   // GB2[6869] := 16#D1C5;
   // GB2[6870] := 16#BCAF;
   // GB2[6871] := 16#B9CD;
   // GB2[6872] := 16#EFF4;
   // GB2[6873] := 16#B4C6;
   // GB2[6874] := 16#D3BA;
   // GB2[6875] := 16#F6C2;
   // GB2[6876] := 16#B3FB;
   // GB2[6877] := 16#F6C3;
   // GB2[6878] := 16#B5F1;
   // GB2[6879] := 16#F6C5;
   // GB2[6880] := 16#D3EA;
   // GB2[6881] := 16#F6A7;
   // GB2[6882] := 16#D1A9;
   // GB2[6883] := 16#F6A9;
   // GB2[6884] := 16#F6A8;
   // GB2[6885] := 16#C1E3;
   // GB2[6886] := 16#C0D7;
   // GB2[6887] := 16#B1A2;
   // GB2[6888] := 16#CEED;
   // GB2[6889] := 16#D0E8;
   // GB2[6890] := 16#F6AB;
   // GB2[6891] := 16#CFF6;
   // GB2[6892] := 16#F6AA;
   // GB2[6893] := 16#D5F0;
   // GB2[6894] := 16#F6AC;
   // GB2[6895] := 16#C3B9;
   // GB2[6896] := 16#BBF4;
   // GB2[6897] := 16#F6AE;
   // GB2[6898] := 16#F6AD;
   // GB2[6899] := 16#C4DE;
   // GB2[6900] := 16#C1D8;
   // GB2[6901] := 16#CBAA;
   // GB2[6902] := 16#CFBC;
   // GB2[6903] := 16#F6AF;
   // GB2[6904] := 16#F6B0;
   // GB2[6905] := 16#F6B1;
   // GB2[6906] := 16#C2B6;
   // GB2[6907] := 16#B0D4;
   // GB2[6908] := 16#C5F9;
   // GB2[6909] := 16#F6B2;
   // GB2[6910] := 16#C7E0;
   // GB2[6911] := 16#F6A6;
   // GB2[6912] := 16#BEB8;
   // GB2[6913] := 16#BEB2;
   // GB2[6914] := 16#B5E5;
   // GB2[6915] := 16#B7C7;
   // GB2[6916] := 16#BFBF;
   // GB2[6917] := 16#C3D2;
   // GB2[6918] := 16#C3E6;
   // GB2[6919] := 16#D8CC;
   // GB2[6920] := 16#B8EF;
   // GB2[6921] := 16#BDF9;
   // GB2[6922] := 16#D1A5;
   // GB2[6923] := 16#B0D0;
   // GB2[6924] := 16#F7B0;
   // GB2[6925] := 16#F7B1;
   // GB2[6926] := 16#D0AC;
   // GB2[6927] := 16#B0B0;
   // GB2[6928] := 16#F7B2;
   // GB2[6929] := 16#F7B3;
   // GB2[6930] := 16#F7B4;
   // GB2[6931] := 16#C7CA;
   // GB2[6932] := 16#BECF;
   // GB2[6933] := 16#F7B7;
   // GB2[6934] := 16#F7B6;
   // GB2[6935] := 16#B1DE;
   // GB2[6936] := 16#F7B5;
   // GB2[6937] := 16#F7B8;
   // GB2[6938] := 16#F7B9;
   // GB2[6939] := 16#CEA4;
   // GB2[6940] := 16#C8CD;
   // GB2[6941] := 16#BAAB;
   // GB2[6942] := 16#E8B8;
   // GB2[6943] := 16#E8B9;
   // GB2[6944] := 16#E8BA;
   // GB2[6945] := 16#BEC2;
   // GB2[6946] := 16#D2F4;
   // GB2[6947] := 16#D4CF;
   // GB2[6948] := 16#C9D8;
   // GB2[6949] := 16#D2B3;
   // GB2[6950] := 16#B6A5;
   // GB2[6951] := 16#C7EA;
   // GB2[6952] := 16#F1FC;
   // GB2[6953] := 16#CFEE;
   // GB2[6954] := 16#CBB3;
   // GB2[6955] := 16#D0EB;
   // GB2[6956] := 16#E7EF;
   // GB2[6957] := 16#CDE7;
   // GB2[6958] := 16#B9CB;
   // GB2[6959] := 16#B6D9;
   // GB2[6960] := 16#F1FD;
   // GB2[6961] := 16#B0E4;
   // GB2[6962] := 16#CBCC;
   // GB2[6963] := 16#F1FE;
   // GB2[6964] := 16#D4A4;
   // GB2[6965] := 16#C2AD;
   // GB2[6966] := 16#C1EC;
   // GB2[6967] := 16#C6C4;
   // GB2[6968] := 16#BEB1;
   // GB2[6969] := 16#F2A1;
   // GB2[6970] := 16#BCD5;
   // GB2[6971] := 16#F2A2;
   // GB2[6972] := 16#F2A3;
   // GB2[6973] := 16#F2A4;
   // GB2[6974] := 16#D2C3;
   // GB2[6975] := 16#C6B5;
   // GB2[6976] := 16#CDC7;
   // GB2[6977] := 16#F2A5;
   // GB2[6978] := 16#D3B1;
   // GB2[6979] := 16#BFC5;
   // GB2[6980] := 16#CCE2;
   // GB2[6981] := 16#F2A6;
   // GB2[6982] := 16#F2A7;
   // GB2[6983] := 16#D1D5;
   // GB2[6984] := 16#B6EE;
   // GB2[6985] := 16#F2A8;
   // GB2[6986] := 16#F2A9;
   // GB2[6987] := 16#B5DF;
   // GB2[6988] := 16#F2AA;
   // GB2[6989] := 16#F2AB;
   // GB2[6990] := 16#B2FC;
   // GB2[6991] := 16#F2AC;
   // GB2[6992] := 16#F2AD;
   // GB2[6993] := 16#C8A7;
   // GB2[6994] := 16#B7E7;
   // GB2[6995] := 16#ECA9;
   // GB2[6996] := 16#ECAA;
   // GB2[6997] := 16#ECAB;
   // GB2[6998] := 16#ECAC;
   // GB2[6999] := 16#C6AE;
   // GB2[7000] := 16#ECAD;
   // GB2[7001] := 16#ECAE;
   // GB2[7002] := 16#B7C9;
   // GB2[7003] := 16#CAB3;
   // GB2[7004] := 16#E2B8;
   // GB2[7005] := 16#F7CF;
   // GB2[7006] := 16#F7D0;
   // GB2[7007] := 16#B2CD;
   // GB2[7008] := 16#F7D1;
   // GB2[7009] := 16#F7D3;
   // GB2[7010] := 16#F7D2;
   // GB2[7011] := 16#E2BB;
   // GB2[7012] := 16#BCA2;
   // GB2[7013] := 16#E2BC;
   // GB2[7014] := 16#E2BD;
   // GB2[7015] := 16#E2BE;
   // GB2[7016] := 16#E2BF;
   // GB2[7017] := 16#E2C0;
   // GB2[7018] := 16#E2C1;
   // GB2[7019] := 16#B7B9;
   // GB2[7020] := 16#D2FB;
   // GB2[7021] := 16#BDA4;
   // GB2[7022] := 16#CACE;
   // GB2[7023] := 16#B1A5;
   // GB2[7024] := 16#CBC7;
   // GB2[7025] := 16#E2C2;
   // GB2[7026] := 16#B6FC;
   // GB2[7027] := 16#C8C4;
   // GB2[7028] := 16#E2C3;
   // GB2[7029] := 16#BDC8;
   // GB2[7030] := 16#B1FD;
   // GB2[7031] := 16#E2C4;
   // GB2[7032] := 16#B6F6;
   // GB2[7033] := 16#E2C5;
   // GB2[7034] := 16#C4D9;
   // GB2[7035] := 16#E2C6;
   // GB2[7036] := 16#CFDA;
   // GB2[7037] := 16#B9DD;
   // GB2[7038] := 16#E2C7;
   // GB2[7039] := 16#C0A1;
   // GB2[7040] := 16#E2C8;
   // GB2[7041] := 16#B2F6;
   // GB2[7042] := 16#E2C9;
   // GB2[7043] := 16#C1F3;
   // GB2[7044] := 16#E2CA;
   // GB2[7045] := 16#E2CB;
   // GB2[7046] := 16#C2F8;
   // GB2[7047] := 16#E2CC;
   // GB2[7048] := 16#E2CD;
   // GB2[7049] := 16#E2CE;
   // GB2[7050] := 16#CAD7;
   // GB2[7051] := 16#D8B8;
   // GB2[7052] := 16#D9E5;
   // GB2[7053] := 16#CFE3;
   // GB2[7054] := 16#F0A5;
   // GB2[7055] := 16#DCB0;
   // GB2[7056] := 16#C2ED;
   // GB2[7057] := 16#D4A6;
   // GB2[7058] := 16#CDD4;
   // GB2[7059] := 16#D1B1;
   // GB2[7060] := 16#B3DB;
   // GB2[7061] := 16#C7FD;
   // GB2[7062] := 16#B2B5;
   // GB2[7063] := 16#C2BF;
   // GB2[7064] := 16#E6E0;
   // GB2[7065] := 16#CABB;
   // GB2[7066] := 16#E6E1;
   // GB2[7067] := 16#E6E2;
   // GB2[7068] := 16#BED4;
   // GB2[7069] := 16#E6E3;
   // GB2[7070] := 16#D7A4;
   // GB2[7071] := 16#CDD5;
   // GB2[7072] := 16#E6E5;
   // GB2[7073] := 16#BCDD;
   // GB2[7074] := 16#E6E4;
   // GB2[7075] := 16#E6E6;
   // GB2[7076] := 16#E6E7;
   // GB2[7077] := 16#C2EE;
   // GB2[7078] := 16#BDBE;
   // GB2[7079] := 16#E6E8;
   // GB2[7080] := 16#C2E6;
   // GB2[7081] := 16#BAA7;
   // GB2[7082] := 16#E6E9;
   // GB2[7083] := 16#E6EA;
   // GB2[7084] := 16#B3D2;
   // GB2[7085] := 16#D1E9;
   // GB2[7086] := 16#BFA5;
   // GB2[7087] := 16#E6EB;
   // GB2[7088] := 16#C6EF;
   // GB2[7089] := 16#E6EC;
   // GB2[7090] := 16#E6ED;
   // GB2[7091] := 16#E6EE;
   // GB2[7092] := 16#C6AD;
   // GB2[7093] := 16#E6EF;
   // GB2[7094] := 16#C9A7;
   // GB2[7095] := 16#E6F0;
   // GB2[7096] := 16#E6F1;
   // GB2[7097] := 16#E6F2;
   // GB2[7098] := 16#E5B9;
   // GB2[7099] := 16#E6F3;
   // GB2[7100] := 16#E6F4;
   // GB2[7101] := 16#C2E2;
   // GB2[7102] := 16#E6F5;
   // GB2[7103] := 16#E6F6;
   // GB2[7104] := 16#D6E8;
   // GB2[7105] := 16#E6F7;
   // GB2[7106] := 16#E6F8;
   // GB2[7107] := 16#B9C7;
   // GB2[7108] := 16#F7BB;
   // GB2[7109] := 16#F7BA;
   // GB2[7110] := 16#F7BE;
   // GB2[7111] := 16#F7BC;
   // GB2[7112] := 16#BAA1;
   // GB2[7113] := 16#F7BF;
   // GB2[7114] := 16#F7C0;
   // GB2[7115] := 16#F7C2;
   // GB2[7116] := 16#F7C1;
   // GB2[7117] := 16#F7C4;
   // GB2[7118] := 16#F7C3;
   // GB2[7119] := 16#F7C5;
   // GB2[7120] := 16#F7C6;
   // GB2[7121] := 16#F7C7;
   // GB2[7122] := 16#CBE8;
   // GB2[7123] := 16#B8DF;
   // GB2[7124] := 16#F7D4;
   // GB2[7125] := 16#F7D5;
   // GB2[7126] := 16#F7D6;
   // GB2[7127] := 16#F7D8;
   // GB2[7128] := 16#F7DA;
   // GB2[7129] := 16#F7D7;
   // GB2[7130] := 16#F7DB;
   // GB2[7131] := 16#F7D9;
   // GB2[7132] := 16#D7D7;
   // GB2[7133] := 16#F7DC;
   // GB2[7134] := 16#F7DD;
   // GB2[7135] := 16#F7DE;
   // GB2[7136] := 16#F7DF;
   // GB2[7137] := 16#F7E0;
   // GB2[7138] := 16#DBCB;
   // GB2[7139] := 16#D8AA;
   // GB2[7140] := 16#E5F7;
   // GB2[7141] := 16#B9ED;
   // GB2[7142] := 16#BFFD;
   // GB2[7143] := 16#BBEA;
   // GB2[7144] := 16#F7C9;
   // GB2[7145] := 16#C6C7;
   // GB2[7146] := 16#F7C8;
   // GB2[7147] := 16#F7CA;
   // GB2[7148] := 16#F7CC;
   // GB2[7149] := 16#F7CB;
   // GB2[7150] := 16#F7CD;
   // GB2[7151] := 16#CEBA;
   // GB2[7152] := 16#F7CE;
   // GB2[7153] := 16#C4A7;
   // GB2[7154] := 16#D3E3;
   // GB2[7155] := 16#F6CF;
   // GB2[7156] := 16#C2B3;
   // GB2[7157] := 16#F6D0;
   // GB2[7158] := 16#F6D1;
   // GB2[7159] := 16#F6D2;
   // GB2[7160] := 16#F6D3;
   // GB2[7161] := 16#F6D4;
   // GB2[7162] := 16#F6D6;
   // GB2[7163] := 16#B1AB;
   // GB2[7164] := 16#F6D7;
   // GB2[7165] := 16#F6D8;
   // GB2[7166] := 16#F6D9;
   // GB2[7167] := 16#F6DA;
   // GB2[7168] := 16#F6DB;
   // GB2[7169] := 16#F6DC;
   // GB2[7170] := 16#F6DD;
   // GB2[7171] := 16#F6DE;
   // GB2[7172] := 16#CFCA;
   // GB2[7173] := 16#F6DF;
   // GB2[7174] := 16#F6E0;
   // GB2[7175] := 16#F6E1;
   // GB2[7176] := 16#F6E2;
   // GB2[7177] := 16#F6E3;
   // GB2[7178] := 16#F6E4;
   // GB2[7179] := 16#C0F0;
   // GB2[7180] := 16#F6E5;
   // GB2[7181] := 16#F6E6;
   // GB2[7182] := 16#F6E7;
   // GB2[7183] := 16#F6E8;
   // GB2[7184] := 16#F6E9;
   // GB2[7185] := 16#F6EA;
   // GB2[7186] := 16#F6EB;
   // GB2[7187] := 16#F6EC;
   // GB2[7188] := 16#F6ED;
   // GB2[7189] := 16#F6EE;
   // GB2[7190] := 16#F6EF;
   // GB2[7191] := 16#F6F0;
   // GB2[7192] := 16#F6F1;
   // GB2[7193] := 16#F6F2;
   // GB2[7194] := 16#F6F3;
   // GB2[7195] := 16#F6F4;
   // GB2[7196] := 16#BEA8;
   // GB2[7197] := 16#F6F5;
   // GB2[7198] := 16#F6F6;
   // GB2[7199] := 16#F6F7;
   // GB2[7200] := 16#F6F8;
   // GB2[7201] := 16#C8FA;
   // GB2[7202] := 16#F6F9;
   // GB2[7203] := 16#F6FA;
   // GB2[7204] := 16#F6FB;
   // GB2[7205] := 16#F6FC;
   // GB2[7206] := 16#F6FD;
   // GB2[7207] := 16#F6FE;
   // GB2[7208] := 16#F7A1;
   // GB2[7209] := 16#F7A2;
   // GB2[7210] := 16#F7A3;
   // GB2[7211] := 16#F7A4;
   // GB2[7212] := 16#F7A5;
   // GB2[7213] := 16#F7A6;
   // GB2[7214] := 16#F7A7;
   // GB2[7215] := 16#F7A8;
   // GB2[7216] := 16#B1EE;
   // GB2[7217] := 16#F7A9;
   // GB2[7218] := 16#F7AA;
   // GB2[7219] := 16#F7AB;
   // GB2[7220] := 16#F7AC;
   // GB2[7221] := 16#F7AD;
   // GB2[7222] := 16#C1DB;
   // GB2[7223] := 16#F7AE;
   // GB2[7224] := 16#F7AF;
   // GB2[7225] := 16#C4F1;
   // GB2[7226] := 16#F0AF;
   // GB2[7227] := 16#BCA6;
   // GB2[7228] := 16#F0B0;
   // GB2[7229] := 16#C3F9;
   // GB2[7230] := 16#C5B8;
   // GB2[7231] := 16#D1BB;
   // GB2[7232] := 16#F0B1;
   // GB2[7233] := 16#F0B2;
   // GB2[7234] := 16#F0B3;
   // GB2[7235] := 16#F0B4;
   // GB2[7236] := 16#F0B5;
   // GB2[7237] := 16#D1BC;
   // GB2[7238] := 16#D1EC;
   // GB2[7239] := 16#F0B7;
   // GB2[7240] := 16#F0B6;
   // GB2[7241] := 16#D4A7;
   // GB2[7242] := 16#CDD2;
   // GB2[7243] := 16#F0B8;
   // GB2[7244] := 16#F0BA;
   // GB2[7245] := 16#F0B9;
   // GB2[7246] := 16#F0BB;
   // GB2[7247] := 16#F0BC;
   // GB2[7248] := 16#B8EB;
   // GB2[7249] := 16#F0BD;
   // GB2[7250] := 16#BAE8;
   // GB2[7251] := 16#F0BE;
   // GB2[7252] := 16#F0BF;
   // GB2[7253] := 16#BEE9;
   // GB2[7254] := 16#F0C0;
   // GB2[7255] := 16#B6EC;
   // GB2[7256] := 16#F0C1;
   // GB2[7257] := 16#F0C2;
   // GB2[7258] := 16#F0C3;
   // GB2[7259] := 16#F0C4;
   // GB2[7260] := 16#C8B5;
   // GB2[7261] := 16#F0C5;
   // GB2[7262] := 16#F0C6;
   // GB2[7263] := 16#F0C7;
   // GB2[7264] := 16#C5F4;
   // GB2[7265] := 16#F0C8;
   // GB2[7266] := 16#F0C9;
   // GB2[7267] := 16#F0CA;
   // GB2[7268] := 16#F7BD;
   // GB2[7269] := 16#F0CB;
   // GB2[7270] := 16#F0CC;
   // GB2[7271] := 16#F0CD;
   // GB2[7272] := 16#F0CE;
   // GB2[7273] := 16#F0CF;
   // GB2[7274] := 16#BAD7;
   // GB2[7275] := 16#F0D0;
   // GB2[7276] := 16#F0D1;
   // GB2[7277] := 16#F0D2;
   // GB2[7278] := 16#F0D3;
   // GB2[7279] := 16#F0D4;
   // GB2[7280] := 16#F0D5;
   // GB2[7281] := 16#F0D6;
   // GB2[7282] := 16#F0D8;
   // GB2[7283] := 16#D3A5;
   // GB2[7284] := 16#F0D7;
   // GB2[7285] := 16#F0D9;
   // GB2[7286] := 16#F5BA;
   // GB2[7287] := 16#C2B9;
   // GB2[7288] := 16#F7E4;
   // GB2[7289] := 16#F7E5;
   // GB2[7290] := 16#F7E6;
   // GB2[7291] := 16#F7E7;
   // GB2[7292] := 16#F7E8;
   // GB2[7293] := 16#C2B4;
   // GB2[7294] := 16#F7EA;
   // GB2[7295] := 16#F7EB;
   // GB2[7296] := 16#C2F3;
   // GB2[7297] := 16#F4F0;
   // GB2[7298] := 16#F4EF;
   // GB2[7299] := 16#C2E9;
   // GB2[7300] := 16#F7E1;
   // GB2[7301] := 16#F7E2;
   // GB2[7302] := 16#BBC6;
   // GB2[7303] := 16#D9E4;
   // GB2[7304] := 16#CAF2;
   // GB2[7305] := 16#C0E8;
   // GB2[7306] := 16#F0A4;
   // GB2[7307] := 16#BADA;
   // GB2[7308] := 16#C7AD;
   // GB2[7309] := 16#C4AC;
   // GB2[7310] := 16#F7EC;
   // GB2[7311] := 16#F7ED;
   // GB2[7312] := 16#F7EE;
   // GB2[7313] := 16#F7F0;
   // GB2[7314] := 16#F7EF;
   // GB2[7315] := 16#F7F1;
   // GB2[7316] := 16#F7F4;
   // GB2[7317] := 16#F7F3;
   // GB2[7318] := 16#F7F2;
   // GB2[7319] := 16#F7F5;
   // GB2[7320] := 16#F7F6;
   // GB2[7321] := 16#EDE9;
   // GB2[7322] := 16#EDEA;
   // GB2[7323] := 16#EDEB;
   // GB2[7324] := 16#F6BC;
   // GB2[7325] := 16#F6BD;
   // GB2[7326] := 16#F6BE;
   // GB2[7327] := 16#B6A6;
   // GB2[7328] := 16#D8BE;
   // GB2[7329] := 16#B9C4;
   // GB2[7330] := 16#D8BB;
   // GB2[7331] := 16#DCB1;
   // GB2[7332] := 16#CAF3;
   // GB2[7333] := 16#F7F7;
   // GB2[7334] := 16#F7F8;
   // GB2[7335] := 16#F7F9;
   // GB2[7336] := 16#F7FB;
   // GB2[7337] := 16#F7FA;
   // GB2[7338] := 16#B1C7;
   // GB2[7339] := 16#F7FC;
   // GB2[7340] := 16#F7FD;
   // GB2[7341] := 16#F7FE;
   // GB2[7342] := 16#C6EB;
   // GB2[7343] := 16#ECB4;
   // GB2[7344] := 16#B3DD;
   // GB2[7345] := 16#F6B3;
   // GB2[7346] := 16#F6B4;
   // GB2[7347] := 16#C1E4;
   // GB2[7348] := 16#F6B5;
   // GB2[7349] := 16#F6B6;
   // GB2[7350] := 16#F6B7;
   // GB2[7351] := 16#F6B8;
   // GB2[7352] := 16#F6B9;
   // GB2[7353] := 16#F6BA;
   // GB2[7354] := 16#C8A3;
   // GB2[7355] := 16#F6BB;
   // GB2[7356] := 16#C1FA;
   // GB2[7357] := 16#B9A8;
   // GB2[7358] := 16#EDE8;
   // GB2[7359] := 16#B9EA;
   // GB2[7360] := 16#D9DF;
   // GB2[7361] := 16#A6F2;
   // GB2[7362] := 16#A6F4;
   // GB2[7363] := 16#A6F5;
   // GB2[7364] := 16#A6E0;
   // GB2[7365] := 16#A6E1;
   // GB2[7366] := 16#A6F0;
   // GB2[7367] := 16#A6F1;
   // GB2[7368] := 16#A6E2;
   // GB2[7369] := 16#A6E3;
   // GB2[7370] := 16#A6EE;
   // GB2[7371] := 16#A6EF;
   // GB2[7372] := 16#A6E6;
   // GB2[7373] := 16#A6E7;
   // GB2[7374] := 16#A6E4;
   // GB2[7375] := 16#A6E5;
   // GB2[7376] := 16#A6E8;
   // GB2[7377] := 16#A6E9;
   // GB2[7378] := 16#A6EA;
   // GB2[7379] := 16#A6EB;
   // GB2[7380] := 16#A3A1;
   // GB2[7381] := 16#A3A2;
   // GB2[7382] := 16#A3A3;
   // GB2[7383] := 16#A1E7;
   // GB2[7384] := 16#A3A5;
   // GB2[7385] := 16#A3A6;
   // GB2[7386] := 16#A3A7;
   // GB2[7387] := 16#A3A8;
   // GB2[7388] := 16#A3A9;
   // GB2[7389] := 16#A3AA;
   // GB2[7390] := 16#A3AB;
   // GB2[7391] := 16#A3AC;
   // GB2[7392] := 16#A3AD;
   // GB2[7393] := 16#A3AE;
   // GB2[7394] := 16#A3AF;
   // GB2[7395] := 16#A3B0;
   // GB2[7396] := 16#A3B1;
   // GB2[7397] := 16#A3B2;
   // GB2[7398] := 16#A3B3;
   // GB2[7399] := 16#A3B4;
   // GB2[7400] := 16#A3B5;
   // GB2[7401] := 16#A3B6;
   // GB2[7402] := 16#A3B7;
   // GB2[7403] := 16#A3B8;
   // GB2[7404] := 16#A3B9;
   // GB2[7405] := 16#A3BA;
   // GB2[7406] := 16#A3BB;
   // GB2[7407] := 16#A3BC;
   // GB2[7408] := 16#A3BD;
   // GB2[7409] := 16#A3BE;
   // GB2[7410] := 16#A3BF;
   // GB2[7411] := 16#A3C0;
   // GB2[7412] := 16#A3C1;
   // GB2[7413] := 16#A3C2;
   // GB2[7414] := 16#A3C3;
   // GB2[7415] := 16#A3C4;
   // GB2[7416] := 16#A3C5;
   // GB2[7417] := 16#A3C6;
   // GB2[7418] := 16#A3C7;
   // GB2[7419] := 16#A3C8;
   // GB2[7420] := 16#A3C9;
   // GB2[7421] := 16#A3CA;
   // GB2[7422] := 16#A3CB;
   // GB2[7423] := 16#A3CC;
   // GB2[7424] := 16#A3CD;
   // GB2[7425] := 16#A3CE;
   // GB2[7426] := 16#A3CF;
   // GB2[7427] := 16#A3D0;
   // GB2[7428] := 16#A3D1;
   // GB2[7429] := 16#A3D2;
   // GB2[7430] := 16#A3D3;
   // GB2[7431] := 16#A3D4;
   // GB2[7432] := 16#A3D5;
   // GB2[7433] := 16#A3D6;
   // GB2[7434] := 16#A3D7;
   // GB2[7435] := 16#A3D8;
   // GB2[7436] := 16#A3D9;
   // GB2[7437] := 16#A3DA;
   // GB2[7438] := 16#A3DB;
   // GB2[7439] := 16#A3DC;
   // GB2[7440] := 16#A3DD;
   // GB2[7441] := 16#A3DE;
   // GB2[7442] := 16#A3DF;
   // GB2[7443] := 16#A3E0;
   // GB2[7444] := 16#A3E1;
   // GB2[7445] := 16#A3E2;
   // GB2[7446] := 16#A3E3;
   // GB2[7447] := 16#A3E4;
   // GB2[7448] := 16#A3E5;
   // GB2[7449] := 16#A3E6;
   // GB2[7450] := 16#A3E7;
   // GB2[7451] := 16#A3E8;
   // GB2[7452] := 16#A3E9;
   // GB2[7453] := 16#A3EA;
   // GB2[7454] := 16#A3EB;
   // GB2[7455] := 16#A3EC;
   // GB2[7456] := 16#A3ED;
   // GB2[7457] := 16#A3EE;
   // GB2[7458] := 16#A3EF;
   // GB2[7459] := 16#A3F0;
   // GB2[7460] := 16#A3F1;
   // GB2[7461] := 16#A3F2;
   // GB2[7462] := 16#A3F3;
   // GB2[7463] := 16#A3F4;
   // GB2[7464] := 16#A3F5;
   // GB2[7465] := 16#A3F6;
   // GB2[7466] := 16#A3F7;
   // GB2[7467] := 16#A3F8;
   // GB2[7468] := 16#A3F9;
   // GB2[7469] := 16#A3FA;
   // GB2[7470] := 16#A3FB;
   // GB2[7471] := 16#A3FC;
   // GB2[7472] := 16#A3FD;
   // GB2[7473] := 16#A1AB;
   // GB2[7474] := 16#A1E9;
   // GB2[7475] := 16#A1EA;
   // GB2[7476] := 16#A3FE;
   // GB2[7477] := 16#A3A4;
   // GB2[7478] := 0;
   // GB2[7479] := 0;
BEGIN
   IF #UNICODE < 16#0080 THEN
       #GB2312 := #UNICODE;
   ELSE
       #hi := 7480;
       #li := 0;
       FOR #j := 0 TO 13 BY 1 DO
           #i := #li + (#hi - #li) / 2;
           IF #UNICODE = #UNI[#i] THEN
               #GB2312 := #GB2[#i];
               EXIT;
           END_IF;
           IF #UNICODE > #UNI[#i] THEN
               #li := #i;
           ELSE
               #hi := #i;
           END_IF;
       END_FOR;
   END_IF;
END_FUNCTION_BLOCK

// ===== library: MasterCopy "UNI_TO_GBK" =====

// folder: FB/UNICODE_FB

FUNCTION_BLOCK "UNI_TO_GBK"   // FB1, SCL
{ S7_Optimized_Access := 'TRUE' }
VERSION : 0.1
   VAR_INPUT
      UNICODE : Word;
   END_VAR
   VAR_OUTPUT
      GBK : Word;
   END_VAR
   VAR
      UNICODE_TO_GBK : Array[0..43592] of Word;
   END_VAR
   VAR_TEMP
      i : UDInt;
      j : UDInt;
      li : UDInt;
      hi : UDInt;
   END_VAR
   // UNICODE_TO_GBK[0] := 16#00A4;
   // UNICODE_TO_GBK[1] := 16#A1E8;
   // UNICODE_TO_GBK[2] := 16#00A7;
   // UNICODE_TO_GBK[3] := 16#A1EC;
   // UNICODE_TO_GBK[4] := 16#00A8;
   // UNICODE_TO_GBK[5] := 16#A1A7;
   // UNICODE_TO_GBK[6] := 16#00B0;
   // UNICODE_TO_GBK[7] := 16#A1E3;
   // UNICODE_TO_GBK[8] := 16#00B1;
   // UNICODE_TO_GBK[9] := 16#A1C0;
   // UNICODE_TO_GBK[10] := 16#00B7;
   // UNICODE_TO_GBK[11] := 16#A1A4;
   // UNICODE_TO_GBK[12] := 16#00D7;
   // UNICODE_TO_GBK[13] := 16#A1C1;
   // UNICODE_TO_GBK[14] := 16#00E0;
   // UNICODE_TO_GBK[15] := 16#A8A4;
   // UNICODE_TO_GBK[16] := 16#00E1;
   // UNICODE_TO_GBK[17] := 16#A8A2;
   // UNICODE_TO_GBK[18] := 16#00E8;
   // UNICODE_TO_GBK[19] := 16#A8A8;
   // UNICODE_TO_GBK[20] := 16#00E9;
   // UNICODE_TO_GBK[21] := 16#A8A6;
   // UNICODE_TO_GBK[22] := 16#00EA;
   // UNICODE_TO_GBK[23] := 16#A8BA;
   // UNICODE_TO_GBK[24] := 16#00EC;
   // UNICODE_TO_GBK[25] := 16#A8AC;
   // UNICODE_TO_GBK[26] := 16#00ED;
   // UNICODE_TO_GBK[27] := 16#A8AA;
   // UNICODE_TO_GBK[28] := 16#00F2;
   // UNICODE_TO_GBK[29] := 16#A8B0;
   // UNICODE_TO_GBK[30] := 16#00F3;
   // UNICODE_TO_GBK[31] := 16#A8AE;
   // UNICODE_TO_GBK[32] := 16#00F7;
   // UNICODE_TO_GBK[33] := 16#A1C2;
   // UNICODE_TO_GBK[34] := 16#00F9;
   // UNICODE_TO_GBK[35] := 16#A8B4;
   // UNICODE_TO_GBK[36] := 16#00FA;
   // UNICODE_TO_GBK[37] := 16#A8B2;
   // UNICODE_TO_GBK[38] := 16#00FC;
   // UNICODE_TO_GBK[39] := 16#A8B9;
   // UNICODE_TO_GBK[40] := 16#0101;
   // UNICODE_TO_GBK[41] := 16#A8A1;
   // UNICODE_TO_GBK[42] := 16#0113;
   // UNICODE_TO_GBK[43] := 16#A8A5;
   // UNICODE_TO_GBK[44] := 16#011B;
   // UNICODE_TO_GBK[45] := 16#A8A7;
   // UNICODE_TO_GBK[46] := 16#012B;
   // UNICODE_TO_GBK[47] := 16#A8A9;
   // UNICODE_TO_GBK[48] := 16#0144;
   // UNICODE_TO_GBK[49] := 16#A8BD;
   // UNICODE_TO_GBK[50] := 16#0148;
   // UNICODE_TO_GBK[51] := 16#A8BE;
   // UNICODE_TO_GBK[52] := 16#014D;
   // UNICODE_TO_GBK[53] := 16#A8AD;
   // UNICODE_TO_GBK[54] := 16#016B;
   // UNICODE_TO_GBK[55] := 16#A8B1;
   // UNICODE_TO_GBK[56] := 16#01CE;
   // UNICODE_TO_GBK[57] := 16#A8A3;
   // UNICODE_TO_GBK[58] := 16#01D0;
   // UNICODE_TO_GBK[59] := 16#A8AB;
   // UNICODE_TO_GBK[60] := 16#01D2;
   // UNICODE_TO_GBK[61] := 16#A8AF;
   // UNICODE_TO_GBK[62] := 16#01D4;
   // UNICODE_TO_GBK[63] := 16#A8B3;
   // UNICODE_TO_GBK[64] := 16#01D6;
   // UNICODE_TO_GBK[65] := 16#A8B5;
   // UNICODE_TO_GBK[66] := 16#01D8;
   // UNICODE_TO_GBK[67] := 16#A8B6;
   // UNICODE_TO_GBK[68] := 16#01DA;
   // UNICODE_TO_GBK[69] := 16#A8B7;
   // UNICODE_TO_GBK[70] := 16#01DC;
   // UNICODE_TO_GBK[71] := 16#A8B8;
   // UNICODE_TO_GBK[72] := 16#0251;
   // UNICODE_TO_GBK[73] := 16#A8BB;
   // UNICODE_TO_GBK[74] := 16#0261;
   // UNICODE_TO_GBK[75] := 16#A8C0;
   // UNICODE_TO_GBK[76] := 16#02C7;
   // UNICODE_TO_GBK[77] := 16#A1A6;
   // UNICODE_TO_GBK[78] := 16#02C9;
   // UNICODE_TO_GBK[79] := 16#A1A5;
   // UNICODE_TO_GBK[80] := 16#02CA;
   // UNICODE_TO_GBK[81] := 16#A840;
   // UNICODE_TO_GBK[82] := 16#02CB;
   // UNICODE_TO_GBK[83] := 16#A841;
   // UNICODE_TO_GBK[84] := 16#02D9;
   // UNICODE_TO_GBK[85] := 16#A842;
   // UNICODE_TO_GBK[86] := 16#0391;
   // UNICODE_TO_GBK[87] := 16#A6A1;
   // UNICODE_TO_GBK[88] := 16#0392;
   // UNICODE_TO_GBK[89] := 16#A6A2;
   // UNICODE_TO_GBK[90] := 16#0393;
   // UNICODE_TO_GBK[91] := 16#A6A3;
   // UNICODE_TO_GBK[92] := 16#0394;
   // UNICODE_TO_GBK[93] := 16#A6A4;
   // UNICODE_TO_GBK[94] := 16#0395;
   // UNICODE_TO_GBK[95] := 16#A6A5;
   // UNICODE_TO_GBK[96] := 16#0396;
   // UNICODE_TO_GBK[97] := 16#A6A6;
   // UNICODE_TO_GBK[98] := 16#0397;
   // UNICODE_TO_GBK[99] := 16#A6A7;
   // UNICODE_TO_GBK[100] := 16#0398;
   // UNICODE_TO_GBK[101] := 16#A6A8;
   // UNICODE_TO_GBK[102] := 16#0399;
   // UNICODE_TO_GBK[103] := 16#A6A9;
   // UNICODE_TO_GBK[104] := 16#039A;
   // UNICODE_TO_GBK[105] := 16#A6AA;
   // UNICODE_TO_GBK[106] := 16#039B;
   // UNICODE_TO_GBK[107] := 16#A6AB;
   // UNICODE_TO_GBK[108] := 16#039C;
   // UNICODE_TO_GBK[109] := 16#A6AC;
   // UNICODE_TO_GBK[110] := 16#039D;
   // UNICODE_TO_GBK[111] := 16#A6AD;
   // UNICODE_TO_GBK[112] := 16#039E;
   // UNICODE_TO_GBK[113] := 16#A6AE;
   // UNICODE_TO_GBK[114] := 16#039F;
   // UNICODE_TO_GBK[115] := 16#A6AF;
   // UNICODE_TO_GBK[116] := 16#03A0;
   // UNICODE_TO_GBK[117] := 16#A6B0;
   // UNICODE_TO_GBK[118] := 16#03A1;
   // UNICODE_TO_GBK[119] := 16#A6B1;
   // UNICODE_TO_GBK[120] := 16#03A3;
   // UNICODE_TO_GBK[121] := 16#A6B2;
   // UNICODE_TO_GBK[122] := 16#03A4;
   // UNICODE_TO_GBK[123] := 16#A6B3;
   // UNICODE_TO_GBK[124] := 16#03A5;
   // UNICODE_TO_GBK[125] := 16#A6B4;
   // UNICODE_TO_GBK[126] := 16#03A6;
   // UNICODE_TO_GBK[127] := 16#A6B5;
   // UNICODE_TO_GBK[128] := 16#03A7;
   // UNICODE_TO_GBK[129] := 16#A6B6;
   // UNICODE_TO_GBK[130] := 16#03A8;
   // UNICODE_TO_GBK[131] := 16#A6B7;
   // UNICODE_TO_GBK[132] := 16#03A9;
   // UNICODE_TO_GBK[133] := 16#A6B8;
   // UNICODE_TO_GBK[134] := 16#03B1;
   // UNICODE_TO_GBK[135] := 16#A6C1;
   // UNICODE_TO_GBK[136] := 16#03B2;
   // UNICODE_TO_GBK[137] := 16#A6C2;
   // UNICODE_TO_GBK[138] := 16#03B3;
   // UNICODE_TO_GBK[139] := 16#A6C3;
   // UNICODE_TO_GBK[140] := 16#03B4;
   // UNICODE_TO_GBK[141] := 16#A6C4;
   // UNICODE_TO_GBK[142] := 16#03B5;
   // UNICODE_TO_GBK[143] := 16#A6C5;
   // UNICODE_TO_GBK[144] := 16#03B6;
   // UNICODE_TO_GBK[145] := 16#A6C6;
   // UNICODE_TO_GBK[146] := 16#03B7;
   // UNICODE_TO_GBK[147] := 16#A6C7;
   // UNICODE_TO_GBK[148] := 16#03B8;
   // UNICODE_TO_GBK[149] := 16#A6C8;
   // UNICODE_TO_GBK[150] := 16#03B9;
   // UNICODE_TO_GBK[151] := 16#A6C9;
   // UNICODE_TO_GBK[152] := 16#03BA;
   // UNICODE_TO_GBK[153] := 16#A6CA;
   // UNICODE_TO_GBK[154] := 16#03BB;
   // UNICODE_TO_GBK[155] := 16#A6CB;
   // UNICODE_TO_GBK[156] := 16#03BC;
   // UNICODE_TO_GBK[157] := 16#A6CC;
   // UNICODE_TO_GBK[158] := 16#03BD;
   // UNICODE_TO_GBK[159] := 16#A6CD;
   // UNICODE_TO_GBK[160] := 16#03BE;
   // UNICODE_TO_GBK[161] := 16#A6CE;
   // UNICODE_TO_GBK[162] := 16#03BF;
   // UNICODE_TO_GBK[163] := 16#A6CF;
   // UNICODE_TO_GBK[164] := 16#03C0;
   // UNICODE_TO_GBK[165] := 16#A6D0;
   // UNICODE_TO_GBK[166] := 16#03C1;
   // UNICODE_TO_GBK[167] := 16#A6D1;
   // UNICODE_TO_GBK[168] := 16#03C3;
   // UNICODE_TO_GBK[169] := 16#A6D2;
   // UNICODE_TO_GBK[170] := 16#03C4;
   // UNICODE_TO_GBK[171] := 16#A6D3;
   // UNICODE_TO_GBK[172] := 16#03C5;
   // UNICODE_TO_GBK[173] := 16#A6D4;
   // UNICODE_TO_GBK[174] := 16#03C6;
   // UNICODE_TO_GBK[175] := 16#A6D5;
   // UNICODE_TO_GBK[176] := 16#03C7;
   // UNICODE_TO_GBK[177] := 16#A6D6;
   // UNICODE_TO_GBK[178] := 16#03C8;
   // UNICODE_TO_GBK[179] := 16#A6D7;
   // UNICODE_TO_GBK[180] := 16#03C9;
   // UNICODE_TO_GBK[181] := 16#A6D8;
   // UNICODE_TO_GBK[182] := 16#0401;
   // UNICODE_TO_GBK[183] := 16#A7A7;
   // UNICODE_TO_GBK[184] := 16#0410;
   // UNICODE_TO_GBK[185] := 16#A7A1;
   // UNICODE_TO_GBK[186] := 16#0411;
   // UNICODE_TO_GBK[187] := 16#A7A2;
   // UNICODE_TO_GBK[188] := 16#0412;
   // UNICODE_TO_GBK[189] := 16#A7A3;
   // UNICODE_TO_GBK[190] := 16#0413;
   // UNICODE_TO_GBK[191] := 16#A7A4;
   // UNICODE_TO_GBK[192] := 16#0414;
   // UNICODE_TO_GBK[193] := 16#A7A5;
   // UNICODE_TO_GBK[194] := 16#0415;
   // UNICODE_TO_GBK[195] := 16#A7A6;
   // UNICODE_TO_GBK[196] := 16#0416;
   // UNICODE_TO_GBK[197] := 16#A7A8;
   // UNICODE_TO_GBK[198] := 16#0417;
   // UNICODE_TO_GBK[199] := 16#A7A9;
   // UNICODE_TO_GBK[200] := 16#0418;
   // UNICODE_TO_GBK[201] := 16#A7AA;
   // UNICODE_TO_GBK[202] := 16#0419;
   // UNICODE_TO_GBK[203] := 16#A7AB;
   // UNICODE_TO_GBK[204] := 16#041A;
   // UNICODE_TO_GBK[205] := 16#A7AC;
   // UNICODE_TO_GBK[206] := 16#041B;
   // UNICODE_TO_GBK[207] := 16#A7AD;
   // UNICODE_TO_GBK[208] := 16#041C;
   // UNICODE_TO_GBK[209] := 16#A7AE;
   // UNICODE_TO_GBK[210] := 16#041D;
   // UNICODE_TO_GBK[211] := 16#A7AF;
   // UNICODE_TO_GBK[212] := 16#041E;
   // UNICODE_TO_GBK[213] := 16#A7B0;
   // UNICODE_TO_GBK[214] := 16#041F;
   // UNICODE_TO_GBK[215] := 16#A7B1;
   // UNICODE_TO_GBK[216] := 16#0420;
   // UNICODE_TO_GBK[217] := 16#A7B2;
   // UNICODE_TO_GBK[218] := 16#0421;
   // UNICODE_TO_GBK[219] := 16#A7B3;
   // UNICODE_TO_GBK[220] := 16#0422;
   // UNICODE_TO_GBK[221] := 16#A7B4;
   // UNICODE_TO_GBK[222] := 16#0423;
   // UNICODE_TO_GBK[223] := 16#A7B5;
   // UNICODE_TO_GBK[224] := 16#0424;
   // UNICODE_TO_GBK[225] := 16#A7B6;
   // UNICODE_TO_GBK[226] := 16#0425;
   // UNICODE_TO_GBK[227] := 16#A7B7;
   // UNICODE_TO_GBK[228] := 16#0426;
   // UNICODE_TO_GBK[229] := 16#A7B8;
   // UNICODE_TO_GBK[230] := 16#0427;
   // UNICODE_TO_GBK[231] := 16#A7B9;
   // UNICODE_TO_GBK[232] := 16#0428;
   // UNICODE_TO_GBK[233] := 16#A7BA;
   // UNICODE_TO_GBK[234] := 16#0429;
   // UNICODE_TO_GBK[235] := 16#A7BB;
   // UNICODE_TO_GBK[236] := 16#042A;
   // UNICODE_TO_GBK[237] := 16#A7BC;
   // UNICODE_TO_GBK[238] := 16#042B;
   // UNICODE_TO_GBK[239] := 16#A7BD;
   // UNICODE_TO_GBK[240] := 16#042C;
   // UNICODE_TO_GBK[241] := 16#A7BE;
   // UNICODE_TO_GBK[242] := 16#042D;
   // UNICODE_TO_GBK[243] := 16#A7BF;
   // UNICODE_TO_GBK[244] := 16#042E;
   // UNICODE_TO_GBK[245] := 16#A7C0;
   // UNICODE_TO_GBK[246] := 16#042F;
   // UNICODE_TO_GBK[247] := 16#A7C1;
   // UNICODE_TO_GBK[248] := 16#0430;
   // UNICODE_TO_GBK[249] := 16#A7D1;
   // UNICODE_TO_GBK[250] := 16#0431;
   // UNICODE_TO_GBK[251] := 16#A7D2;
   // UNICODE_TO_GBK[252] := 16#0432;
   // UNICODE_TO_GBK[253] := 16#A7D3;
   // UNICODE_TO_GBK[254] := 16#0433;
   // UNICODE_TO_GBK[255] := 16#A7D4;
   // UNICODE_TO_GBK[256] := 16#0434;
   // UNICODE_TO_GBK[257] := 16#A7D5;
   // UNICODE_TO_GBK[258] := 16#0435;
   // UNICODE_TO_GBK[259] := 16#A7D6;
   // UNICODE_TO_GBK[260] := 16#0436;
   // UNICODE_TO_GBK[261] := 16#A7D8;
   // UNICODE_TO_GBK[262] := 16#0437;
   // UNICODE_TO_GBK[263] := 16#A7D9;
   // UNICODE_TO_GBK[264] := 16#0438;
   // UNICODE_TO_GBK[265] := 16#A7DA;
   // UNICODE_TO_GBK[266] := 16#0439;
   // UNICODE_TO_GBK[267] := 16#A7DB;
   // UNICODE_TO_GBK[268] := 16#043A;
   // UNICODE_TO_GBK[269] := 16#A7DC;
   // UNICODE_TO_GBK[270] := 16#043B;
   // UNICODE_TO_GBK[271] := 16#A7DD;
   // UNICODE_TO_GBK[272] := 16#043C;
   // UNICODE_TO_GBK[273] := 16#A7DE;
   // UNICODE_TO_GBK[274] := 16#043D;
   // UNICODE_TO_GBK[275] := 16#A7DF;
   // UNICODE_TO_GBK[276] := 16#043E;
   // UNICODE_TO_GBK[277] := 16#A7E0;
   // UNICODE_TO_GBK[278] := 16#043F;
   // UNICODE_TO_GBK[279] := 16#A7E1;
   // UNICODE_TO_GBK[280] := 16#0440;
   // UNICODE_TO_GBK[281] := 16#A7E2;
   // UNICODE_TO_GBK[282] := 16#0441;
   // UNICODE_TO_GBK[283] := 16#A7E3;
   // UNICODE_TO_GBK[284] := 16#0442;
   // UNICODE_TO_GBK[285] := 16#A7E4;
   // UNICODE_TO_GBK[286] := 16#0443;
   // UNICODE_TO_GBK[287] := 16#A7E5;
   // UNICODE_TO_GBK[288] := 16#0444;
   // UNICODE_TO_GBK[289] := 16#A7E6;
   // UNICODE_TO_GBK[290] := 16#0445;
   // UNICODE_TO_GBK[291] := 16#A7E7;
   // UNICODE_TO_GBK[292] := 16#0446;
   // UNICODE_TO_GBK[293] := 16#A7E8;
   // UNICODE_TO_GBK[294] := 16#0447;
   // UNICODE_TO_GBK[295] := 16#A7E9;
   // UNICODE_TO_GBK[296] := 16#0448;
   // UNICODE_TO_GBK[297] := 16#A7EA;
   // UNICODE_TO_GBK[298] := 16#0449;
   // UNICODE_TO_GBK[299] := 16#A7EB;
   // UNICODE_TO_GBK[300] := 16#044A;
   // UNICODE_TO_GBK[301] := 16#A7EC;
   // UNICODE_TO_GBK[302] := 16#044B;
   // UNICODE_TO_GBK[303] := 16#A7ED;
   // UNICODE_TO_GBK[304] := 16#044C;
   // UNICODE_TO_GBK[305] := 16#A7EE;
   // UNICODE_TO_GBK[306] := 16#044D;
   // UNICODE_TO_GBK[307] := 16#A7EF;
   // UNICODE_TO_GBK[308] := 16#044E;
   // UNICODE_TO_GBK[309] := 16#A7F0;
   // UNICODE_TO_GBK[310] := 16#044F;
   // UNICODE_TO_GBK[311] := 16#A7F1;
   // UNICODE_TO_GBK[312] := 16#0451;
   // UNICODE_TO_GBK[313] := 16#A7D7;
   // UNICODE_TO_GBK[314] := 16#2010;
   // UNICODE_TO_GBK[315] := 16#A95C;
   // UNICODE_TO_GBK[316] := 16#2013;
   // UNICODE_TO_GBK[317] := 16#A843;
   // UNICODE_TO_GBK[318] := 16#2014;
   // UNICODE_TO_GBK[319] := 16#A1AA;
   // UNICODE_TO_GBK[320] := 16#2015;
   // UNICODE_TO_GBK[321] := 16#A844;
   // UNICODE_TO_GBK[322] := 16#2016;
   // UNICODE_TO_GBK[323] := 16#A1AC;
   // UNICODE_TO_GBK[324] := 16#2018;
   // UNICODE_TO_GBK[325] := 16#A1AE;
   // UNICODE_TO_GBK[326] := 16#2019;
   // UNICODE_TO_GBK[327] := 16#A1AF;
   // UNICODE_TO_GBK[328] := 16#201C;
   // UNICODE_TO_GBK[329] := 16#A1B0;
   // UNICODE_TO_GBK[330] := 16#201D;
   // UNICODE_TO_GBK[331] := 16#A1B1;
   // UNICODE_TO_GBK[332] := 16#2025;
   // UNICODE_TO_GBK[333] := 16#A845;
   // UNICODE_TO_GBK[334] := 16#2026;
   // UNICODE_TO_GBK[335] := 16#A1AD;
   // UNICODE_TO_GBK[336] := 16#2030;
   // UNICODE_TO_GBK[337] := 16#A1EB;
   // UNICODE_TO_GBK[338] := 16#2032;
   // UNICODE_TO_GBK[339] := 16#A1E4;
   // UNICODE_TO_GBK[340] := 16#2033;
   // UNICODE_TO_GBK[341] := 16#A1E5;
   // UNICODE_TO_GBK[342] := 16#2035;
   // UNICODE_TO_GBK[343] := 16#A846;
   // UNICODE_TO_GBK[344] := 16#203B;
   // UNICODE_TO_GBK[345] := 16#A1F9;
   // UNICODE_TO_GBK[346] := 16#20AC;
   // UNICODE_TO_GBK[347] := 16#0080;
   // UNICODE_TO_GBK[348] := 16#2103;
   // UNICODE_TO_GBK[349] := 16#A1E6;
   // UNICODE_TO_GBK[350] := 16#2105;
   // UNICODE_TO_GBK[351] := 16#A847;
   // UNICODE_TO_GBK[352] := 16#2109;
   // UNICODE_TO_GBK[353] := 16#A848;
   // UNICODE_TO_GBK[354] := 16#2116;
   // UNICODE_TO_GBK[355] := 16#A1ED;
   // UNICODE_TO_GBK[356] := 16#2121;
   // UNICODE_TO_GBK[357] := 16#A959;
   // UNICODE_TO_GBK[358] := 16#2160;
   // UNICODE_TO_GBK[359] := 16#A2F1;
   // UNICODE_TO_GBK[360] := 16#2161;
   // UNICODE_TO_GBK[361] := 16#A2F2;
   // UNICODE_TO_GBK[362] := 16#2162;
   // UNICODE_TO_GBK[363] := 16#A2F3;
   // UNICODE_TO_GBK[364] := 16#2163;
   // UNICODE_TO_GBK[365] := 16#A2F4;
   // UNICODE_TO_GBK[366] := 16#2164;
   // UNICODE_TO_GBK[367] := 16#A2F5;
   // UNICODE_TO_GBK[368] := 16#2165;
   // UNICODE_TO_GBK[369] := 16#A2F6;
   // UNICODE_TO_GBK[370] := 16#2166;
   // UNICODE_TO_GBK[371] := 16#A2F7;
   // UNICODE_TO_GBK[372] := 16#2167;
   // UNICODE_TO_GBK[373] := 16#A2F8;
   // UNICODE_TO_GBK[374] := 16#2168;
   // UNICODE_TO_GBK[375] := 16#A2F9;
   // UNICODE_TO_GBK[376] := 16#2169;
   // UNICODE_TO_GBK[377] := 16#A2FA;
   // UNICODE_TO_GBK[378] := 16#216A;
   // UNICODE_TO_GBK[379] := 16#A2FB;
   // UNICODE_TO_GBK[380] := 16#216B;
   // UNICODE_TO_GBK[381] := 16#A2FC;
   // UNICODE_TO_GBK[382] := 16#2170;
   // UNICODE_TO_GBK[383] := 16#A2A1;
   // UNICODE_TO_GBK[384] := 16#2171;
   // UNICODE_TO_GBK[385] := 16#A2A2;
   // UNICODE_TO_GBK[386] := 16#2172;
   // UNICODE_TO_GBK[387] := 16#A2A3;
   // UNICODE_TO_GBK[388] := 16#2173;
   // UNICODE_TO_GBK[389] := 16#A2A4;
   // UNICODE_TO_GBK[390] := 16#2174;
   // UNICODE_TO_GBK[391] := 16#A2A5;
   // UNICODE_TO_GBK[392] := 16#2175;
   // UNICODE_TO_GBK[393] := 16#A2A6;
   // UNICODE_TO_GBK[394] := 16#2176;
   // UNICODE_TO_GBK[395] := 16#A2A7;
   // UNICODE_TO_GBK[396] := 16#2177;
   // UNICODE_TO_GBK[397] := 16#A2A8;
   // UNICODE_TO_GBK[398] := 16#2178;
   // UNICODE_TO_GBK[399] := 16#A2A9;
   // UNICODE_TO_GBK[400] := 16#2179;
   // UNICODE_TO_GBK[401] := 16#A2AA;
   // UNICODE_TO_GBK[402] := 16#2190;
   // UNICODE_TO_GBK[403] := 16#A1FB;
   // UNICODE_TO_GBK[404] := 16#2191;
   // UNICODE_TO_GBK[405] := 16#A1FC;
   // UNICODE_TO_GBK[406] := 16#2192;
   // UNICODE_TO_GBK[407] := 16#A1FA;
   // UNICODE_TO_GBK[408] := 16#2193;
   // UNICODE_TO_GBK[409] := 16#A1FD;
   // UNICODE_TO_GBK[410] := 16#2196;
   // UNICODE_TO_GBK[411] := 16#A849;
   // UNICODE_TO_GBK[412] := 16#2197;
   // UNICODE_TO_GBK[413] := 16#A84A;
   // UNICODE_TO_GBK[414] := 16#2198;
   // UNICODE_TO_GBK[415] := 16#A84B;
   // UNICODE_TO_GBK[416] := 16#2199;
   // UNICODE_TO_GBK[417] := 16#A84C;
   // UNICODE_TO_GBK[418] := 16#2208;
   // UNICODE_TO_GBK[419] := 16#A1CA;
   // UNICODE_TO_GBK[420] := 16#220F;
   // UNICODE_TO_GBK[421] := 16#A1C7;
   // UNICODE_TO_GBK[422] := 16#2211;
   // UNICODE_TO_GBK[423] := 16#A1C6;
   // UNICODE_TO_GBK[424] := 16#2215;
   // UNICODE_TO_GBK[425] := 16#A84D;
   // UNICODE_TO_GBK[426] := 16#221A;
   // UNICODE_TO_GBK[427] := 16#A1CC;
   // UNICODE_TO_GBK[428] := 16#221D;
   // UNICODE_TO_GBK[429] := 16#A1D8;
   // UNICODE_TO_GBK[430] := 16#221E;
   // UNICODE_TO_GBK[431] := 16#A1DE;
   // UNICODE_TO_GBK[432] := 16#221F;
   // UNICODE_TO_GBK[433] := 16#A84E;
   // UNICODE_TO_GBK[434] := 16#2220;
   // UNICODE_TO_GBK[435] := 16#A1CF;
   // UNICODE_TO_GBK[436] := 16#2223;
   // UNICODE_TO_GBK[437] := 16#A84F;
   // UNICODE_TO_GBK[438] := 16#2225;
   // UNICODE_TO_GBK[439] := 16#A1CE;
   // UNICODE_TO_GBK[440] := 16#2227;
   // UNICODE_TO_GBK[441] := 16#A1C4;
   // UNICODE_TO_GBK[442] := 16#2228;
   // UNICODE_TO_GBK[443] := 16#A1C5;
   // UNICODE_TO_GBK[444] := 16#2229;
   // UNICODE_TO_GBK[445] := 16#A1C9;
   // UNICODE_TO_GBK[446] := 16#222A;
   // UNICODE_TO_GBK[447] := 16#A1C8;
   // UNICODE_TO_GBK[448] := 16#222B;
   // UNICODE_TO_GBK[449] := 16#A1D2;
   // UNICODE_TO_GBK[450] := 16#222E;
   // UNICODE_TO_GBK[451] := 16#A1D3;
   // UNICODE_TO_GBK[452] := 16#2234;
   // UNICODE_TO_GBK[453] := 16#A1E0;
   // UNICODE_TO_GBK[454] := 16#2235;
   // UNICODE_TO_GBK[455] := 16#A1DF;
   // UNICODE_TO_GBK[456] := 16#2236;
   // UNICODE_TO_GBK[457] := 16#A1C3;
   // UNICODE_TO_GBK[458] := 16#2237;
   // UNICODE_TO_GBK[459] := 16#A1CB;
   // UNICODE_TO_GBK[460] := 16#223D;
   // UNICODE_TO_GBK[461] := 16#A1D7;
   // UNICODE_TO_GBK[462] := 16#2248;
   // UNICODE_TO_GBK[463] := 16#A1D6;
   // UNICODE_TO_GBK[464] := 16#224C;
   // UNICODE_TO_GBK[465] := 16#A1D5;
   // UNICODE_TO_GBK[466] := 16#2252;
   // UNICODE_TO_GBK[467] := 16#A850;
   // UNICODE_TO_GBK[468] := 16#2260;
   // UNICODE_TO_GBK[469] := 16#A1D9;
   // UNICODE_TO_GBK[470] := 16#2261;
   // UNICODE_TO_GBK[471] := 16#A1D4;
   // UNICODE_TO_GBK[472] := 16#2264;
   // UNICODE_TO_GBK[473] := 16#A1DC;
   // UNICODE_TO_GBK[474] := 16#2265;
   // UNICODE_TO_GBK[475] := 16#A1DD;
   // UNICODE_TO_GBK[476] := 16#2266;
   // UNICODE_TO_GBK[477] := 16#A851;
   // UNICODE_TO_GBK[478] := 16#2267;
   // UNICODE_TO_GBK[479] := 16#A852;
   // UNICODE_TO_GBK[480] := 16#226E;
   // UNICODE_TO_GBK[481] := 16#A1DA;
   // UNICODE_TO_GBK[482] := 16#226F;
   // UNICODE_TO_GBK[483] := 16#A1DB;
   // UNICODE_TO_GBK[484] := 16#2295;
   // UNICODE_TO_GBK[485] := 16#A892;
   // UNICODE_TO_GBK[486] := 16#2299;
   // UNICODE_TO_GBK[487] := 16#A1D1;
   // UNICODE_TO_GBK[488] := 16#22A5;
   // UNICODE_TO_GBK[489] := 16#A1CD;
   // UNICODE_TO_GBK[490] := 16#22BF;
   // UNICODE_TO_GBK[491] := 16#A853;
   // UNICODE_TO_GBK[492] := 16#2312;
   // UNICODE_TO_GBK[493] := 16#A1D0;
   // UNICODE_TO_GBK[494] := 16#2460;
   // UNICODE_TO_GBK[495] := 16#A2D9;
   // UNICODE_TO_GBK[496] := 16#2461;
   // UNICODE_TO_GBK[497] := 16#A2DA;
   // UNICODE_TO_GBK[498] := 16#2462;
   // UNICODE_TO_GBK[499] := 16#A2DB;
   // UNICODE_TO_GBK[500] := 16#2463;
   // UNICODE_TO_GBK[501] := 16#A2DC;
   // UNICODE_TO_GBK[502] := 16#2464;
   // UNICODE_TO_GBK[503] := 16#A2DD;
   // UNICODE_TO_GBK[504] := 16#2465;
   // UNICODE_TO_GBK[505] := 16#A2DE;
   // UNICODE_TO_GBK[506] := 16#2466;
   // UNICODE_TO_GBK[507] := 16#A2DF;
   // UNICODE_TO_GBK[508] := 16#2467;
   // UNICODE_TO_GBK[509] := 16#A2E0;
   // UNICODE_TO_GBK[510] := 16#2468;
   // UNICODE_TO_GBK[511] := 16#A2E1;
   // UNICODE_TO_GBK[512] := 16#2469;
   // UNICODE_TO_GBK[513] := 16#A2E2;
   // UNICODE_TO_GBK[514] := 16#2474;
   // UNICODE_TO_GBK[515] := 16#A2C5;
   // UNICODE_TO_GBK[516] := 16#2475;
   // UNICODE_TO_GBK[517] := 16#A2C6;
   // UNICODE_TO_GBK[518] := 16#2476;
   // UNICODE_TO_GBK[519] := 16#A2C7;
   // UNICODE_TO_GBK[520] := 16#2477;
   // UNICODE_TO_GBK[521] := 16#A2C8;
   // UNICODE_TO_GBK[522] := 16#2478;
   // UNICODE_TO_GBK[523] := 16#A2C9;
   // UNICODE_TO_GBK[524] := 16#2479;
   // UNICODE_TO_GBK[525] := 16#A2CA;
   // UNICODE_TO_GBK[526] := 16#247A;
   // UNICODE_TO_GBK[527] := 16#A2CB;
   // UNICODE_TO_GBK[528] := 16#247B;
   // UNICODE_TO_GBK[529] := 16#A2CC;
   // UNICODE_TO_GBK[530] := 16#247C;
   // UNICODE_TO_GBK[531] := 16#A2CD;
   // UNICODE_TO_GBK[532] := 16#247D;
   // UNICODE_TO_GBK[533] := 16#A2CE;
   // UNICODE_TO_GBK[534] := 16#247E;
   // UNICODE_TO_GBK[535] := 16#A2CF;
   // UNICODE_TO_GBK[536] := 16#247F;
   // UNICODE_TO_GBK[537] := 16#A2D0;
   // UNICODE_TO_GBK[538] := 16#2480;
   // UNICODE_TO_GBK[539] := 16#A2D1;
   // UNICODE_TO_GBK[540] := 16#2481;
   // UNICODE_TO_GBK[541] := 16#A2D2;
   // UNICODE_TO_GBK[542] := 16#2482;
   // UNICODE_TO_GBK[543] := 16#A2D3;
   // UNICODE_TO_GBK[544] := 16#2483;
   // UNICODE_TO_GBK[545] := 16#A2D4;
   // UNICODE_TO_GBK[546] := 16#2484;
   // UNICODE_TO_GBK[547] := 16#A2D5;
   // UNICODE_TO_GBK[548] := 16#2485;
   // UNICODE_TO_GBK[549] := 16#A2D6;
   // UNICODE_TO_GBK[550] := 16#2486;
   // UNICODE_TO_GBK[551] := 16#A2D7;
   // UNICODE_TO_GBK[552] := 16#2487;
   // UNICODE_TO_GBK[553] := 16#A2D8;
   // UNICODE_TO_GBK[554] := 16#2488;
   // UNICODE_TO_GBK[555] := 16#A2B1;
   // UNICODE_TO_GBK[556] := 16#2489;
   // UNICODE_TO_GBK[557] := 16#A2B2;
   // UNICODE_TO_GBK[558] := 16#248A;
   // UNICODE_TO_GBK[559] := 16#A2B3;
   // UNICODE_TO_GBK[560] := 16#248B;
   // UNICODE_TO_GBK[561] := 16#A2B4;
   // UNICODE_TO_GBK[562] := 16#248C;
   // UNICODE_TO_GBK[563] := 16#A2B5;
   // UNICODE_TO_GBK[564] := 16#248D;
   // UNICODE_TO_GBK[565] := 16#A2B6;
   // UNICODE_TO_GBK[566] := 16#248E;
   // UNICODE_TO_GBK[567] := 16#A2B7;
   // UNICODE_TO_GBK[568] := 16#248F;
   // UNICODE_TO_GBK[569] := 16#A2B8;
   // UNICODE_TO_GBK[570] := 16#2490;
   // UNICODE_TO_GBK[571] := 16#A2B9;
   // UNICODE_TO_GBK[572] := 16#2491;
   // UNICODE_TO_GBK[573] := 16#A2BA;
   // UNICODE_TO_GBK[574] := 16#2492;
   // UNICODE_TO_GBK[575] := 16#A2BB;
   // UNICODE_TO_GBK[576] := 16#2493;
   // UNICODE_TO_GBK[577] := 16#A2BC;
   // UNICODE_TO_GBK[578] := 16#2494;
   // UNICODE_TO_GBK[579] := 16#A2BD;
   // UNICODE_TO_GBK[580] := 16#2495;
   // UNICODE_TO_GBK[581] := 16#A2BE;
   // UNICODE_TO_GBK[582] := 16#2496;
   // UNICODE_TO_GBK[583] := 16#A2BF;
   // UNICODE_TO_GBK[584] := 16#2497;
   // UNICODE_TO_GBK[585] := 16#A2C0;
   // UNICODE_TO_GBK[586] := 16#2498;
   // UNICODE_TO_GBK[587] := 16#A2C1;
   // UNICODE_TO_GBK[588] := 16#2499;
   // UNICODE_TO_GBK[589] := 16#A2C2;
   // UNICODE_TO_GBK[590] := 16#249A;
   // UNICODE_TO_GBK[591] := 16#A2C3;
   // UNICODE_TO_GBK[592] := 16#249B;
   // UNICODE_TO_GBK[593] := 16#A2C4;
   // UNICODE_TO_GBK[594] := 16#2500;
   // UNICODE_TO_GBK[595] := 16#A9A4;
   // UNICODE_TO_GBK[596] := 16#2501;
   // UNICODE_TO_GBK[597] := 16#A9A5;
   // UNICODE_TO_GBK[598] := 16#2502;
   // UNICODE_TO_GBK[599] := 16#A9A6;
   // UNICODE_TO_GBK[600] := 16#2503;
   // UNICODE_TO_GBK[601] := 16#A9A7;
   // UNICODE_TO_GBK[602] := 16#2504;
   // UNICODE_TO_GBK[603] := 16#A9A8;
   // UNICODE_TO_GBK[604] := 16#2505;
   // UNICODE_TO_GBK[605] := 16#A9A9;
   // UNICODE_TO_GBK[606] := 16#2506;
   // UNICODE_TO_GBK[607] := 16#A9AA;
   // UNICODE_TO_GBK[608] := 16#2507;
   // UNICODE_TO_GBK[609] := 16#A9AB;
   // UNICODE_TO_GBK[610] := 16#2508;
   // UNICODE_TO_GBK[611] := 16#A9AC;
   // UNICODE_TO_GBK[612] := 16#2509;
   // UNICODE_TO_GBK[613] := 16#A9AD;
   // UNICODE_TO_GBK[614] := 16#250A;
   // UNICODE_TO_GBK[615] := 16#A9AE;
   // UNICODE_TO_GBK[616] := 16#250B;
   // UNICODE_TO_GBK[617] := 16#A9AF;
   // UNICODE_TO_GBK[618] := 16#250C;
   // UNICODE_TO_GBK[619] := 16#A9B0;
   // UNICODE_TO_GBK[620] := 16#250D;
   // UNICODE_TO_GBK[621] := 16#A9B1;
   // UNICODE_TO_GBK[622] := 16#250E;
   // UNICODE_TO_GBK[623] := 16#A9B2;
   // UNICODE_TO_GBK[624] := 16#250F;
   // UNICODE_TO_GBK[625] := 16#A9B3;
   // UNICODE_TO_GBK[626] := 16#2510;
   // UNICODE_TO_GBK[627] := 16#A9B4;
   // UNICODE_TO_GBK[628] := 16#2511;
   // UNICODE_TO_GBK[629] := 16#A9B5;
   // UNICODE_TO_GBK[630] := 16#2512;
   // UNICODE_TO_GBK[631] := 16#A9B6;
   // UNICODE_TO_GBK[632] := 16#2513;
   // UNICODE_TO_GBK[633] := 16#A9B7;
   // UNICODE_TO_GBK[634] := 16#2514;
   // UNICODE_TO_GBK[635] := 16#A9B8;
   // UNICODE_TO_GBK[636] := 16#2515;
   // UNICODE_TO_GBK[637] := 16#A9B9;
   // UNICODE_TO_GBK[638] := 16#2516;
   // UNICODE_TO_GBK[639] := 16#A9BA;
   // UNICODE_TO_GBK[640] := 16#2517;
   // UNICODE_TO_GBK[641] := 16#A9BB;
   // UNICODE_TO_GBK[642] := 16#2518;
   // UNICODE_TO_GBK[643] := 16#A9BC;
   // UNICODE_TO_GBK[644] := 16#2519;
   // UNICODE_TO_GBK[645] := 16#A9BD;
   // UNICODE_TO_GBK[646] := 16#251A;
   // UNICODE_TO_GBK[647] := 16#A9BE;
   // UNICODE_TO_GBK[648] := 16#251B;
   // UNICODE_TO_GBK[649] := 16#A9BF;
   // UNICODE_TO_GBK[650] := 16#251C;
   // UNICODE_TO_GBK[651] := 16#A9C0;
   // UNICODE_TO_GBK[652] := 16#251D;
   // UNICODE_TO_GBK[653] := 16#A9C1;
   // UNICODE_TO_GBK[654] := 16#251E;
   // UNICODE_TO_GBK[655] := 16#A9C2;
   // UNICODE_TO_GBK[656] := 16#251F;
   // UNICODE_TO_GBK[657] := 16#A9C3;
   // UNICODE_TO_GBK[658] := 16#2520;
   // UNICODE_TO_GBK[659] := 16#A9C4;
   // UNICODE_TO_GBK[660] := 16#2521;
   // UNICODE_TO_GBK[661] := 16#A9C5;
   // UNICODE_TO_GBK[662] := 16#2522;
   // UNICODE_TO_GBK[663] := 16#A9C6;
   // UNICODE_TO_GBK[664] := 16#2523;
   // UNICODE_TO_GBK[665] := 16#A9C7;
   // UNICODE_TO_GBK[666] := 16#2524;
   // UNICODE_TO_GBK[667] := 16#A9C8;
   // UNICODE_TO_GBK[668] := 16#2525;
   // UNICODE_TO_GBK[669] := 16#A9C9;
   // UNICODE_TO_GBK[670] := 16#2526;
   // UNICODE_TO_GBK[671] := 16#A9CA;
   // UNICODE_TO_GBK[672] := 16#2527;
   // UNICODE_TO_GBK[673] := 16#A9CB;
   // UNICODE_TO_GBK[674] := 16#2528;
   // UNICODE_TO_GBK[675] := 16#A9CC;
   // UNICODE_TO_GBK[676] := 16#2529;
   // UNICODE_TO_GBK[677] := 16#A9CD;
   // UNICODE_TO_GBK[678] := 16#252A;
   // UNICODE_TO_GBK[679] := 16#A9CE;
   // UNICODE_TO_GBK[680] := 16#252B;
   // UNICODE_TO_GBK[681] := 16#A9CF;
   // UNICODE_TO_GBK[682] := 16#252C;
   // UNICODE_TO_GBK[683] := 16#A9D0;
   // UNICODE_TO_GBK[684] := 16#252D;
   // UNICODE_TO_GBK[685] := 16#A9D1;
   // UNICODE_TO_GBK[686] := 16#252E;
   // UNICODE_TO_GBK[687] := 16#A9D2;
   // UNICODE_TO_GBK[688] := 16#252F;
   // UNICODE_TO_GBK[689] := 16#A9D3;
   // UNICODE_TO_GBK[690] := 16#2530;
   // UNICODE_TO_GBK[691] := 16#A9D4;
   // UNICODE_TO_GBK[692] := 16#2531;
   // UNICODE_TO_GBK[693] := 16#A9D5;
   // UNICODE_TO_GBK[694] := 16#2532;
   // UNICODE_TO_GBK[695] := 16#A9D6;
   // UNICODE_TO_GBK[696] := 16#2533;
   // UNICODE_TO_GBK[697] := 16#A9D7;
   // UNICODE_TO_GBK[698] := 16#2534;
   // UNICODE_TO_GBK[699] := 16#A9D8;
   // UNICODE_TO_GBK[700] := 16#2535;
   // UNICODE_TO_GBK[701] := 16#A9D9;
   // UNICODE_TO_GBK[702] := 16#2536;
   // UNICODE_TO_GBK[703] := 16#A9DA;
   // UNICODE_TO_GBK[704] := 16#2537;
   // UNICODE_TO_GBK[705] := 16#A9DB;
   // UNICODE_TO_GBK[706] := 16#2538;
   // UNICODE_TO_GBK[707] := 16#A9DC;
   // UNICODE_TO_GBK[708] := 16#2539;
   // UNICODE_TO_GBK[709] := 16#A9DD;
   // UNICODE_TO_GBK[710] := 16#253A;
   // UNICODE_TO_GBK[711] := 16#A9DE;
   // UNICODE_TO_GBK[712] := 16#253B;
   // UNICODE_TO_GBK[713] := 16#A9DF;
   // UNICODE_TO_GBK[714] := 16#253C;
   // UNICODE_TO_GBK[715] := 16#A9E0;
   // UNICODE_TO_GBK[716] := 16#253D;
   // UNICODE_TO_GBK[717] := 16#A9E1;
   // UNICODE_TO_GBK[718] := 16#253E;
   // UNICODE_TO_GBK[719] := 16#A9E2;
   // UNICODE_TO_GBK[720] := 16#253F;
   // UNICODE_TO_GBK[721] := 16#A9E3;
   // UNICODE_TO_GBK[722] := 16#2540;
   // UNICODE_TO_GBK[723] := 16#A9E4;
   // UNICODE_TO_GBK[724] := 16#2541;
   // UNICODE_TO_GBK[725] := 16#A9E5;
   // UNICODE_TO_GBK[726] := 16#2542;
   // UNICODE_TO_GBK[727] := 16#A9E6;
   // UNICODE_TO_GBK[728] := 16#2543;
   // UNICODE_TO_GBK[729] := 16#A9E7;
   // UNICODE_TO_GBK[730] := 16#2544;
   // UNICODE_TO_GBK[731] := 16#A9E8;
   // UNICODE_TO_GBK[732] := 16#2545;
   // UNICODE_TO_GBK[733] := 16#A9E9;
   // UNICODE_TO_GBK[734] := 16#2546;
   // UNICODE_TO_GBK[735] := 16#A9EA;
   // UNICODE_TO_GBK[736] := 16#2547;
   // UNICODE_TO_GBK[737] := 16#A9EB;
   // UNICODE_TO_GBK[738] := 16#2548;
   // UNICODE_TO_GBK[739] := 16#A9EC;
   // UNICODE_TO_GBK[740] := 16#2549;
   // UNICODE_TO_GBK[741] := 16#A9ED;
   // UNICODE_TO_GBK[742] := 16#254A;
   // UNICODE_TO_GBK[743] := 16#A9EE;
   // UNICODE_TO_GBK[744] := 16#254B;
   // UNICODE_TO_GBK[745] := 16#A9EF;
   // UNICODE_TO_GBK[746] := 16#2550;
   // UNICODE_TO_GBK[747] := 16#A854;
   // UNICODE_TO_GBK[748] := 16#2551;
   // UNICODE_TO_GBK[749] := 16#A855;
   // UNICODE_TO_GBK[750] := 16#2552;
   // UNICODE_TO_GBK[751] := 16#A856;
   // UNICODE_TO_GBK[752] := 16#2553;
   // UNICODE_TO_GBK[753] := 16#A857;
   // UNICODE_TO_GBK[754] := 16#2554;
   // UNICODE_TO_GBK[755] := 16#A858;
   // UNICODE_TO_GBK[756] := 16#2555;
   // UNICODE_TO_GBK[757] := 16#A859;
   // UNICODE_TO_GBK[758] := 16#2556;
   // UNICODE_TO_GBK[759] := 16#A85A;
   // UNICODE_TO_GBK[760] := 16#2557;
   // UNICODE_TO_GBK[761] := 16#A85B;
   // UNICODE_TO_GBK[762] := 16#2558;
   // UNICODE_TO_GBK[763] := 16#A85C;
   // UNICODE_TO_GBK[764] := 16#2559;
   // UNICODE_TO_GBK[765] := 16#A85D;
   // UNICODE_TO_GBK[766] := 16#255A;
   // UNICODE_TO_GBK[767] := 16#A85E;
   // UNICODE_TO_GBK[768] := 16#255B;
   // UNICODE_TO_GBK[769] := 16#A85F;
   // UNICODE_TO_GBK[770] := 16#255C;
   // UNICODE_TO_GBK[771] := 16#A860;
   // UNICODE_TO_GBK[772] := 16#255D;
   // UNICODE_TO_GBK[773] := 16#A861;
   // UNICODE_TO_GBK[774] := 16#255E;
   // UNICODE_TO_GBK[775] := 16#A862;
   // UNICODE_TO_GBK[776] := 16#255F;
   // UNICODE_TO_GBK[777] := 16#A863;
   // UNICODE_TO_GBK[778] := 16#2560;
   // UNICODE_TO_GBK[779] := 16#A864;
   // UNICODE_TO_GBK[780] := 16#2561;
   // UNICODE_TO_GBK[781] := 16#A865;
   // UNICODE_TO_GBK[782] := 16#2562;
   // UNICODE_TO_GBK[783] := 16#A866;
   // UNICODE_TO_GBK[784] := 16#2563;
   // UNICODE_TO_GBK[785] := 16#A867;
   // UNICODE_TO_GBK[786] := 16#2564;
   // UNICODE_TO_GBK[787] := 16#A868;
   // UNICODE_TO_GBK[788] := 16#2565;
   // UNICODE_TO_GBK[789] := 16#A869;
   // UNICODE_TO_GBK[790] := 16#2566;
   // UNICODE_TO_GBK[791] := 16#A86A;
   // UNICODE_TO_GBK[792] := 16#2567;
   // UNICODE_TO_GBK[793] := 16#A86B;
   // UNICODE_TO_GBK[794] := 16#2568;
   // UNICODE_TO_GBK[795] := 16#A86C;
   // UNICODE_TO_GBK[796] := 16#2569;
   // UNICODE_TO_GBK[797] := 16#A86D;
   // UNICODE_TO_GBK[798] := 16#256A;
   // UNICODE_TO_GBK[799] := 16#A86E;
   // UNICODE_TO_GBK[800] := 16#256B;
   // UNICODE_TO_GBK[801] := 16#A86F;
   // UNICODE_TO_GBK[802] := 16#256C;
   // UNICODE_TO_GBK[803] := 16#A870;
   // UNICODE_TO_GBK[804] := 16#256D;
   // UNICODE_TO_GBK[805] := 16#A871;
   // UNICODE_TO_GBK[806] := 16#256E;
   // UNICODE_TO_GBK[807] := 16#A872;
   // UNICODE_TO_GBK[808] := 16#256F;
   // UNICODE_TO_GBK[809] := 16#A873;
   // UNICODE_TO_GBK[810] := 16#2570;
   // UNICODE_TO_GBK[811] := 16#A874;
   // UNICODE_TO_GBK[812] := 16#2571;
   // UNICODE_TO_GBK[813] := 16#A875;
   // UNICODE_TO_GBK[814] := 16#2572;
   // UNICODE_TO_GBK[815] := 16#A876;
   // UNICODE_TO_GBK[816] := 16#2573;
   // UNICODE_TO_GBK[817] := 16#A877;
   // UNICODE_TO_GBK[818] := 16#2581;
   // UNICODE_TO_GBK[819] := 16#A878;
   // UNICODE_TO_GBK[820] := 16#2582;
   // UNICODE_TO_GBK[821] := 16#A879;
   // UNICODE_TO_GBK[822] := 16#2583;
   // UNICODE_TO_GBK[823] := 16#A87A;
   // UNICODE_TO_GBK[824] := 16#2584;
   // UNICODE_TO_GBK[825] := 16#A87B;
   // UNICODE_TO_GBK[826] := 16#2585;
   // UNICODE_TO_GBK[827] := 16#A87C;
   // UNICODE_TO_GBK[828] := 16#2586;
   // UNICODE_TO_GBK[829] := 16#A87D;
   // UNICODE_TO_GBK[830] := 16#2587;
   // UNICODE_TO_GBK[831] := 16#A87E;
   // UNICODE_TO_GBK[832] := 16#2588;
   // UNICODE_TO_GBK[833] := 16#A880;
   // UNICODE_TO_GBK[834] := 16#2589;
   // UNICODE_TO_GBK[835] := 16#A881;
   // UNICODE_TO_GBK[836] := 16#258A;
   // UNICODE_TO_GBK[837] := 16#A882;
   // UNICODE_TO_GBK[838] := 16#258B;
   // UNICODE_TO_GBK[839] := 16#A883;
   // UNICODE_TO_GBK[840] := 16#258C;
   // UNICODE_TO_GBK[841] := 16#A884;
   // UNICODE_TO_GBK[842] := 16#258D;
   // UNICODE_TO_GBK[843] := 16#A885;
   // UNICODE_TO_GBK[844] := 16#258E;
   // UNICODE_TO_GBK[845] := 16#A886;
   // UNICODE_TO_GBK[846] := 16#258F;
   // UNICODE_TO_GBK[847] := 16#A887;
   // UNICODE_TO_GBK[848] := 16#2593;
   // UNICODE_TO_GBK[849] := 16#A888;
   // UNICODE_TO_GBK[850] := 16#2594;
   // UNICODE_TO_GBK[851] := 16#A889;
   // UNICODE_TO_GBK[852] := 16#2595;
   // UNICODE_TO_GBK[853] := 16#A88A;
   // UNICODE_TO_GBK[854] := 16#25A0;
   // UNICODE_TO_GBK[855] := 16#A1F6;
   // UNICODE_TO_GBK[856] := 16#25A1;
   // UNICODE_TO_GBK[857] := 16#A1F5;
   // UNICODE_TO_GBK[858] := 16#25B2;
   // UNICODE_TO_GBK[859] := 16#A1F8;
   // UNICODE_TO_GBK[860] := 16#25B3;
   // UNICODE_TO_GBK[861] := 16#A1F7;
   // UNICODE_TO_GBK[862] := 16#25BC;
   // UNICODE_TO_GBK[863] := 16#A88B;
   // UNICODE_TO_GBK[864] := 16#25BD;
   // UNICODE_TO_GBK[865] := 16#A88C;
   // UNICODE_TO_GBK[866] := 16#25C6;
   // UNICODE_TO_GBK[867] := 16#A1F4;
   // UNICODE_TO_GBK[868] := 16#25C7;
   // UNICODE_TO_GBK[869] := 16#A1F3;
   // UNICODE_TO_GBK[870] := 16#25CB;
   // UNICODE_TO_GBK[871] := 16#A1F0;
   // UNICODE_TO_GBK[872] := 16#25CE;
   // UNICODE_TO_GBK[873] := 16#A1F2;
   // UNICODE_TO_GBK[874] := 16#25CF;
   // UNICODE_TO_GBK[875] := 16#A1F1;
   // UNICODE_TO_GBK[876] := 16#25E2;
   // UNICODE_TO_GBK[877] := 16#A88D;
   // UNICODE_TO_GBK[878] := 16#25E3;
   // UNICODE_TO_GBK[879] := 16#A88E;
   // UNICODE_TO_GBK[880] := 16#25E4;
   // UNICODE_TO_GBK[881] := 16#A88F;
   // UNICODE_TO_GBK[882] := 16#25E5;
   // UNICODE_TO_GBK[883] := 16#A890;
   // UNICODE_TO_GBK[884] := 16#2605;
   // UNICODE_TO_GBK[885] := 16#A1EF;
   // UNICODE_TO_GBK[886] := 16#2606;
   // UNICODE_TO_GBK[887] := 16#A1EE;
   // UNICODE_TO_GBK[888] := 16#2609;
   // UNICODE_TO_GBK[889] := 16#A891;
   // UNICODE_TO_GBK[890] := 16#2640;
   // UNICODE_TO_GBK[891] := 16#A1E2;
   // UNICODE_TO_GBK[892] := 16#2642;
   // UNICODE_TO_GBK[893] := 16#A1E1;
   // UNICODE_TO_GBK[894] := 16#3000;
   // UNICODE_TO_GBK[895] := 16#A1A1;
   // UNICODE_TO_GBK[896] := 16#3001;
   // UNICODE_TO_GBK[897] := 16#A1A2;
   // UNICODE_TO_GBK[898] := 16#3002;
   // UNICODE_TO_GBK[899] := 16#A1A3;
   // UNICODE_TO_GBK[900] := 16#3003;
   // UNICODE_TO_GBK[901] := 16#A1A8;
   // UNICODE_TO_GBK[902] := 16#3005;
   // UNICODE_TO_GBK[903] := 16#A1A9;
   // UNICODE_TO_GBK[904] := 16#3006;
   // UNICODE_TO_GBK[905] := 16#A965;
   // UNICODE_TO_GBK[906] := 16#3007;
   // UNICODE_TO_GBK[907] := 16#A996;
   // UNICODE_TO_GBK[908] := 16#3008;
   // UNICODE_TO_GBK[909] := 16#A1B4;
   // UNICODE_TO_GBK[910] := 16#3009;
   // UNICODE_TO_GBK[911] := 16#A1B5;
   // UNICODE_TO_GBK[912] := 16#300A;
   // UNICODE_TO_GBK[913] := 16#A1B6;
   // UNICODE_TO_GBK[914] := 16#300B;
   // UNICODE_TO_GBK[915] := 16#A1B7;
   // UNICODE_TO_GBK[916] := 16#300C;
   // UNICODE_TO_GBK[917] := 16#A1B8;
   // UNICODE_TO_GBK[918] := 16#300D;
   // UNICODE_TO_GBK[919] := 16#A1B9;
   // UNICODE_TO_GBK[920] := 16#300E;
   // UNICODE_TO_GBK[921] := 16#A1BA;
   // UNICODE_TO_GBK[922] := 16#300F;
   // UNICODE_TO_GBK[923] := 16#A1BB;
   // UNICODE_TO_GBK[924] := 16#3010;
   // UNICODE_TO_GBK[925] := 16#A1BE;
   // UNICODE_TO_GBK[926] := 16#3011;
   // UNICODE_TO_GBK[927] := 16#A1BF;
   // UNICODE_TO_GBK[928] := 16#3012;
   // UNICODE_TO_GBK[929] := 16#A893;
   // UNICODE_TO_GBK[930] := 16#3013;
   // UNICODE_TO_GBK[931] := 16#A1FE;
   // UNICODE_TO_GBK[932] := 16#3014;
   // UNICODE_TO_GBK[933] := 16#A1B2;
   // UNICODE_TO_GBK[934] := 16#3015;
   // UNICODE_TO_GBK[935] := 16#A1B3;
   // UNICODE_TO_GBK[936] := 16#3016;
   // UNICODE_TO_GBK[937] := 16#A1BC;
   // UNICODE_TO_GBK[938] := 16#3017;
   // UNICODE_TO_GBK[939] := 16#A1BD;
   // UNICODE_TO_GBK[940] := 16#301D;
   // UNICODE_TO_GBK[941] := 16#A894;
   // UNICODE_TO_GBK[942] := 16#301E;
   // UNICODE_TO_GBK[943] := 16#A895;
   // UNICODE_TO_GBK[944] := 16#3021;
   // UNICODE_TO_GBK[945] := 16#A940;
   // UNICODE_TO_GBK[946] := 16#3022;
   // UNICODE_TO_GBK[947] := 16#A941;
   // UNICODE_TO_GBK[948] := 16#3023;
   // UNICODE_TO_GBK[949] := 16#A942;
   // UNICODE_TO_GBK[950] := 16#3024;
   // UNICODE_TO_GBK[951] := 16#A943;
   // UNICODE_TO_GBK[952] := 16#3025;
   // UNICODE_TO_GBK[953] := 16#A944;
   // UNICODE_TO_GBK[954] := 16#3026;
   // UNICODE_TO_GBK[955] := 16#A945;
   // UNICODE_TO_GBK[956] := 16#3027;
   // UNICODE_TO_GBK[957] := 16#A946;
   // UNICODE_TO_GBK[958] := 16#3028;
   // UNICODE_TO_GBK[959] := 16#A947;
   // UNICODE_TO_GBK[960] := 16#3029;
   // UNICODE_TO_GBK[961] := 16#A948;
   // UNICODE_TO_GBK[962] := 16#3041;
   // UNICODE_TO_GBK[963] := 16#A4A1;
   // UNICODE_TO_GBK[964] := 16#3042;
   // UNICODE_TO_GBK[965] := 16#A4A2;
   // UNICODE_TO_GBK[966] := 16#3043;
   // UNICODE_TO_GBK[967] := 16#A4A3;
   // UNICODE_TO_GBK[968] := 16#3044;
   // UNICODE_TO_GBK[969] := 16#A4A4;
   // UNICODE_TO_GBK[970] := 16#3045;
   // UNICODE_TO_GBK[971] := 16#A4A5;
   // UNICODE_TO_GBK[972] := 16#3046;
   // UNICODE_TO_GBK[973] := 16#A4A6;
   // UNICODE_TO_GBK[974] := 16#3047;
   // UNICODE_TO_GBK[975] := 16#A4A7;
   // UNICODE_TO_GBK[976] := 16#3048;
   // UNICODE_TO_GBK[977] := 16#A4A8;
   // UNICODE_TO_GBK[978] := 16#3049;
   // UNICODE_TO_GBK[979] := 16#A4A9;
   // UNICODE_TO_GBK[980] := 16#304A;
   // UNICODE_TO_GBK[981] := 16#A4AA;
   // UNICODE_TO_GBK[982] := 16#304B;
   // UNICODE_TO_GBK[983] := 16#A4AB;
   // UNICODE_TO_GBK[984] := 16#304C;
   // UNICODE_TO_GBK[985] := 16#A4AC;
   // UNICODE_TO_GBK[986] := 16#304D;
   // UNICODE_TO_GBK[987] := 16#A4AD;
   // UNICODE_TO_GBK[988] := 16#304E;
   // UNICODE_TO_GBK[989] := 16#A4AE;
   // UNICODE_TO_GBK[990] := 16#304F;
   // UNICODE_TO_GBK[991] := 16#A4AF;
   // UNICODE_TO_GBK[992] := 16#3050;
   // UNICODE_TO_GBK[993] := 16#A4B0;
   // UNICODE_TO_GBK[994] := 16#3051;
   // UNICODE_TO_GBK[995] := 16#A4B1;
   // UNICODE_TO_GBK[996] := 16#3052;
   // UNICODE_TO_GBK[997] := 16#A4B2;
   // UNICODE_TO_GBK[998] := 16#3053;
   // UNICODE_TO_GBK[999] := 16#A4B3;
   // UNICODE_TO_GBK[1000] := 16#3054;
   // UNICODE_TO_GBK[1001] := 16#A4B4;
   // UNICODE_TO_GBK[1002] := 16#3055;
   // UNICODE_TO_GBK[1003] := 16#A4B5;
   // UNICODE_TO_GBK[1004] := 16#3056;
   // UNICODE_TO_GBK[1005] := 16#A4B6;
   // UNICODE_TO_GBK[1006] := 16#3057;
   // UNICODE_TO_GBK[1007] := 16#A4B7;
   // UNICODE_TO_GBK[1008] := 16#3058;
   // UNICODE_TO_GBK[1009] := 16#A4B8;
   // UNICODE_TO_GBK[1010] := 16#3059;
   // UNICODE_TO_GBK[1011] := 16#A4B9;
   // UNICODE_TO_GBK[1012] := 16#305A;
   // UNICODE_TO_GBK[1013] := 16#A4BA;
   // UNICODE_TO_GBK[1014] := 16#305B;
   // UNICODE_TO_GBK[1015] := 16#A4BB;
   // UNICODE_TO_GBK[1016] := 16#305C;
   // UNICODE_TO_GBK[1017] := 16#A4BC;
   // UNICODE_TO_GBK[1018] := 16#305D;
   // UNICODE_TO_GBK[1019] := 16#A4BD;
   // UNICODE_TO_GBK[1020] := 16#305E;
   // UNICODE_TO_GBK[1021] := 16#A4BE;
   // UNICODE_TO_GBK[1022] := 16#305F;
   // UNICODE_TO_GBK[1023] := 16#A4BF;
   // UNICODE_TO_GBK[1024] := 16#3060;
   // UNICODE_TO_GBK[1025] := 16#A4C0;
   // UNICODE_TO_GBK[1026] := 16#3061;
   // UNICODE_TO_GBK[1027] := 16#A4C1;
   // UNICODE_TO_GBK[1028] := 16#3062;
   // UNICODE_TO_GBK[1029] := 16#A4C2;
   // UNICODE_TO_GBK[1030] := 16#3063;
   // UNICODE_TO_GBK[1031] := 16#A4C3;
   // UNICODE_TO_GBK[1032] := 16#3064;
   // UNICODE_TO_GBK[1033] := 16#A4C4;
   // UNICODE_TO_GBK[1034] := 16#3065;
   // UNICODE_TO_GBK[1035] := 16#A4C5;
   // UNICODE_TO_GBK[1036] := 16#3066;
   // UNICODE_TO_GBK[1037] := 16#A4C6;
   // UNICODE_TO_GBK[1038] := 16#3067;
   // UNICODE_TO_GBK[1039] := 16#A4C7;
   // UNICODE_TO_GBK[1040] := 16#3068;
   // UNICODE_TO_GBK[1041] := 16#A4C8;
   // UNICODE_TO_GBK[1042] := 16#3069;
   // UNICODE_TO_GBK[1043] := 16#A4C9;
   // UNICODE_TO_GBK[1044] := 16#306A;
   // UNICODE_TO_GBK[1045] := 16#A4CA;
   // UNICODE_TO_GBK[1046] := 16#306B;
   // UNICODE_TO_GBK[1047] := 16#A4CB;
   // UNICODE_TO_GBK[1048] := 16#306C;
   // UNICODE_TO_GBK[1049] := 16#A4CC;
   // UNICODE_TO_GBK[1050] := 16#306D;
   // UNICODE_TO_GBK[1051] := 16#A4CD;
   // UNICODE_TO_GBK[1052] := 16#306E;
   // UNICODE_TO_GBK[1053] := 16#A4CE;
   // UNICODE_TO_GBK[1054] := 16#306F;
   // UNICODE_TO_GBK[1055] := 16#A4CF;
   // UNICODE_TO_GBK[1056] := 16#3070;
   // UNICODE_TO_GBK[1057] := 16#A4D0;
   // UNICODE_TO_GBK[1058] := 16#3071;
   // UNICODE_TO_GBK[1059] := 16#A4D1;
   // UNICODE_TO_GBK[1060] := 16#3072;
   // UNICODE_TO_GBK[1061] := 16#A4D2;
   // UNICODE_TO_GBK[1062] := 16#3073;
   // UNICODE_TO_GBK[1063] := 16#A4D3;
   // UNICODE_TO_GBK[1064] := 16#3074;
   // UNICODE_TO_GBK[1065] := 16#A4D4;
   // UNICODE_TO_GBK[1066] := 16#3075;
   // UNICODE_TO_GBK[1067] := 16#A4D5;
   // UNICODE_TO_GBK[1068] := 16#3076;
   // UNICODE_TO_GBK[1069] := 16#A4D6;
   // UNICODE_TO_GBK[1070] := 16#3077;
   // UNICODE_TO_GBK[1071] := 16#A4D7;
   // UNICODE_TO_GBK[1072] := 16#3078;
   // UNICODE_TO_GBK[1073] := 16#A4D8;
   // UNICODE_TO_GBK[1074] := 16#3079;
   // UNICODE_TO_GBK[1075] := 16#A4D9;
   // UNICODE_TO_GBK[1076] := 16#307A;
   // UNICODE_TO_GBK[1077] := 16#A4DA;
   // UNICODE_TO_GBK[1078] := 16#307B;
   // UNICODE_TO_GBK[1079] := 16#A4DB;
   // UNICODE_TO_GBK[1080] := 16#307C;
   // UNICODE_TO_GBK[1081] := 16#A4DC;
   // UNICODE_TO_GBK[1082] := 16#307D;
   // UNICODE_TO_GBK[1083] := 16#A4DD;
   // UNICODE_TO_GBK[1084] := 16#307E;
   // UNICODE_TO_GBK[1085] := 16#A4DE;
   // UNICODE_TO_GBK[1086] := 16#307F;
   // UNICODE_TO_GBK[1087] := 16#A4DF;
   // UNICODE_TO_GBK[1088] := 16#3080;
   // UNICODE_TO_GBK[1089] := 16#A4E0;
   // UNICODE_TO_GBK[1090] := 16#3081;
   // UNICODE_TO_GBK[1091] := 16#A4E1;
   // UNICODE_TO_GBK[1092] := 16#3082;
   // UNICODE_TO_GBK[1093] := 16#A4E2;
   // UNICODE_TO_GBK[1094] := 16#3083;
   // UNICODE_TO_GBK[1095] := 16#A4E3;
   // UNICODE_TO_GBK[1096] := 16#3084;
   // UNICODE_TO_GBK[1097] := 16#A4E4;
   // UNICODE_TO_GBK[1098] := 16#3085;
   // UNICODE_TO_GBK[1099] := 16#A4E5;
   // UNICODE_TO_GBK[1100] := 16#3086;
   // UNICODE_TO_GBK[1101] := 16#A4E6;
   // UNICODE_TO_GBK[1102] := 16#3087;
   // UNICODE_TO_GBK[1103] := 16#A4E7;
   // UNICODE_TO_GBK[1104] := 16#3088;
   // UNICODE_TO_GBK[1105] := 16#A4E8;
   // UNICODE_TO_GBK[1106] := 16#3089;
   // UNICODE_TO_GBK[1107] := 16#A4E9;
   // UNICODE_TO_GBK[1108] := 16#308A;
   // UNICODE_TO_GBK[1109] := 16#A4EA;
   // UNICODE_TO_GBK[1110] := 16#308B;
   // UNICODE_TO_GBK[1111] := 16#A4EB;
   // UNICODE_TO_GBK[1112] := 16#308C;
   // UNICODE_TO_GBK[1113] := 16#A4EC;
   // UNICODE_TO_GBK[1114] := 16#308D;
   // UNICODE_TO_GBK[1115] := 16#A4ED;
   // UNICODE_TO_GBK[1116] := 16#308E;
   // UNICODE_TO_GBK[1117] := 16#A4EE;
   // UNICODE_TO_GBK[1118] := 16#308F;
   // UNICODE_TO_GBK[1119] := 16#A4EF;
   // UNICODE_TO_GBK[1120] := 16#3090;
   // UNICODE_TO_GBK[1121] := 16#A4F0;
   // UNICODE_TO_GBK[1122] := 16#3091;
   // UNICODE_TO_GBK[1123] := 16#A4F1;
   // UNICODE_TO_GBK[1124] := 16#3092;
   // UNICODE_TO_GBK[1125] := 16#A4F2;
   // UNICODE_TO_GBK[1126] := 16#3093;
   // UNICODE_TO_GBK[1127] := 16#A4F3;
   // UNICODE_TO_GBK[1128] := 16#309B;
   // UNICODE_TO_GBK[1129] := 16#A961;
   // UNICODE_TO_GBK[1130] := 16#309C;
   // UNICODE_TO_GBK[1131] := 16#A962;
   // UNICODE_TO_GBK[1132] := 16#309D;
   // UNICODE_TO_GBK[1133] := 16#A966;
   // UNICODE_TO_GBK[1134] := 16#309E;
   // UNICODE_TO_GBK[1135] := 16#A967;
   // UNICODE_TO_GBK[1136] := 16#30A1;
   // UNICODE_TO_GBK[1137] := 16#A5A1;
   // UNICODE_TO_GBK[1138] := 16#30A2;
   // UNICODE_TO_GBK[1139] := 16#A5A2;
   // UNICODE_TO_GBK[1140] := 16#30A3;
   // UNICODE_TO_GBK[1141] := 16#A5A3;
   // UNICODE_TO_GBK[1142] := 16#30A4;
   // UNICODE_TO_GBK[1143] := 16#A5A4;
   // UNICODE_TO_GBK[1144] := 16#30A5;
   // UNICODE_TO_GBK[1145] := 16#A5A5;
   // UNICODE_TO_GBK[1146] := 16#30A6;
   // UNICODE_TO_GBK[1147] := 16#A5A6;
   // UNICODE_TO_GBK[1148] := 16#30A7;
   // UNICODE_TO_GBK[1149] := 16#A5A7;
   // UNICODE_TO_GBK[1150] := 16#30A8;
   // UNICODE_TO_GBK[1151] := 16#A5A8;
   // UNICODE_TO_GBK[1152] := 16#30A9;
   // UNICODE_TO_GBK[1153] := 16#A5A9;
   // UNICODE_TO_GBK[1154] := 16#30AA;
   // UNICODE_TO_GBK[1155] := 16#A5AA;
   // UNICODE_TO_GBK[1156] := 16#30AB;
   // UNICODE_TO_GBK[1157] := 16#A5AB;
   // UNICODE_TO_GBK[1158] := 16#30AC;
   // UNICODE_TO_GBK[1159] := 16#A5AC;
   // UNICODE_TO_GBK[1160] := 16#30AD;
   // UNICODE_TO_GBK[1161] := 16#A5AD;
   // UNICODE_TO_GBK[1162] := 16#30AE;
   // UNICODE_TO_GBK[1163] := 16#A5AE;
   // UNICODE_TO_GBK[1164] := 16#30AF;
   // UNICODE_TO_GBK[1165] := 16#A5AF;
   // UNICODE_TO_GBK[1166] := 16#30B0;
   // UNICODE_TO_GBK[1167] := 16#A5B0;
   // UNICODE_TO_GBK[1168] := 16#30B1;
   // UNICODE_TO_GBK[1169] := 16#A5B1;
   // UNICODE_TO_GBK[1170] := 16#30B2;
   // UNICODE_TO_GBK[1171] := 16#A5B2;
   // UNICODE_TO_GBK[1172] := 16#30B3;
   // UNICODE_TO_GBK[1173] := 16#A5B3;
   // UNICODE_TO_GBK[1174] := 16#30B4;
   // UNICODE_TO_GBK[1175] := 16#A5B4;
   // UNICODE_TO_GBK[1176] := 16#30B5;
   // UNICODE_TO_GBK[1177] := 16#A5B5;
   // UNICODE_TO_GBK[1178] := 16#30B6;
   // UNICODE_TO_GBK[1179] := 16#A5B6;
   // UNICODE_TO_GBK[1180] := 16#30B7;
   // UNICODE_TO_GBK[1181] := 16#A5B7;
   // UNICODE_TO_GBK[1182] := 16#30B8;
   // UNICODE_TO_GBK[1183] := 16#A5B8;
   // UNICODE_TO_GBK[1184] := 16#30B9;
   // UNICODE_TO_GBK[1185] := 16#A5B9;
   // UNICODE_TO_GBK[1186] := 16#30BA;
   // UNICODE_TO_GBK[1187] := 16#A5BA;
   // UNICODE_TO_GBK[1188] := 16#30BB;
   // UNICODE_TO_GBK[1189] := 16#A5BB;
   // UNICODE_TO_GBK[1190] := 16#30BC;
   // UNICODE_TO_GBK[1191] := 16#A5BC;
   // UNICODE_TO_GBK[1192] := 16#30BD;
   // UNICODE_TO_GBK[1193] := 16#A5BD;
   // UNICODE_TO_GBK[1194] := 16#30BE;
   // UNICODE_TO_GBK[1195] := 16#A5BE;
   // UNICODE_TO_GBK[1196] := 16#30BF;
   // UNICODE_TO_GBK[1197] := 16#A5BF;
   // UNICODE_TO_GBK[1198] := 16#30C0;
   // UNICODE_TO_GBK[1199] := 16#A5C0;
   // UNICODE_TO_GBK[1200] := 16#30C1;
   // UNICODE_TO_GBK[1201] := 16#A5C1;
   // UNICODE_TO_GBK[1202] := 16#30C2;
   // UNICODE_TO_GBK[1203] := 16#A5C2;
   // UNICODE_TO_GBK[1204] := 16#30C3;
   // UNICODE_TO_GBK[1205] := 16#A5C3;
   // UNICODE_TO_GBK[1206] := 16#30C4;
   // UNICODE_TO_GBK[1207] := 16#A5C4;
   // UNICODE_TO_GBK[1208] := 16#30C5;
   // UNICODE_TO_GBK[1209] := 16#A5C5;
   // UNICODE_TO_GBK[1210] := 16#30C6;
   // UNICODE_TO_GBK[1211] := 16#A5C6;
   // UNICODE_TO_GBK[1212] := 16#30C7;
   // UNICODE_TO_GBK[1213] := 16#A5C7;
   // UNICODE_TO_GBK[1214] := 16#30C8;
   // UNICODE_TO_GBK[1215] := 16#A5C8;
   // UNICODE_TO_GBK[1216] := 16#30C9;
   // UNICODE_TO_GBK[1217] := 16#A5C9;
   // UNICODE_TO_GBK[1218] := 16#30CA;
   // UNICODE_TO_GBK[1219] := 16#A5CA;
   // UNICODE_TO_GBK[1220] := 16#30CB;
   // UNICODE_TO_GBK[1221] := 16#A5CB;
   // UNICODE_TO_GBK[1222] := 16#30CC;
   // UNICODE_TO_GBK[1223] := 16#A5CC;
   // UNICODE_TO_GBK[1224] := 16#30CD;
   // UNICODE_TO_GBK[1225] := 16#A5CD;
   // UNICODE_TO_GBK[1226] := 16#30CE;
   // UNICODE_TO_GBK[1227] := 16#A5CE;
   // UNICODE_TO_GBK[1228] := 16#30CF;
   // UNICODE_TO_GBK[1229] := 16#A5CF;
   // UNICODE_TO_GBK[1230] := 16#30D0;
   // UNICODE_TO_GBK[1231] := 16#A5D0;
   // UNICODE_TO_GBK[1232] := 16#30D1;
   // UNICODE_TO_GBK[1233] := 16#A5D1;
   // UNICODE_TO_GBK[1234] := 16#30D2;
   // UNICODE_TO_GBK[1235] := 16#A5D2;
   // UNICODE_TO_GBK[1236] := 16#30D3;
   // UNICODE_TO_GBK[1237] := 16#A5D3;
   // UNICODE_TO_GBK[1238] := 16#30D4;
   // UNICODE_TO_GBK[1239] := 16#A5D4;
   // UNICODE_TO_GBK[1240] := 16#30D5;
   // UNICODE_TO_GBK[1241] := 16#A5D5;
   // UNICODE_TO_GBK[1242] := 16#30D6;
   // UNICODE_TO_GBK[1243] := 16#A5D6;
   // UNICODE_TO_GBK[1244] := 16#30D7;
   // UNICODE_TO_GBK[1245] := 16#A5D7;
   // UNICODE_TO_GBK[1246] := 16#30D8;
   // UNICODE_TO_GBK[1247] := 16#A5D8;
   // UNICODE_TO_GBK[1248] := 16#30D9;
   // UNICODE_TO_GBK[1249] := 16#A5D9;
   // UNICODE_TO_GBK[1250] := 16#30DA;
   // UNICODE_TO_GBK[1251] := 16#A5DA;
   // UNICODE_TO_GBK[1252] := 16#30DB;
   // UNICODE_TO_GBK[1253] := 16#A5DB;
   // UNICODE_TO_GBK[1254] := 16#30DC;
   // UNICODE_TO_GBK[1255] := 16#A5DC;
   // UNICODE_TO_GBK[1256] := 16#30DD;
   // UNICODE_TO_GBK[1257] := 16#A5DD;
   // UNICODE_TO_GBK[1258] := 16#30DE;
   // UNICODE_TO_GBK[1259] := 16#A5DE;
   // UNICODE_TO_GBK[1260] := 16#30DF;
   // UNICODE_TO_GBK[1261] := 16#A5DF;
   // UNICODE_TO_GBK[1262] := 16#30E0;
   // UNICODE_TO_GBK[1263] := 16#A5E0;
   // UNICODE_TO_GBK[1264] := 16#30E1;
   // UNICODE_TO_GBK[1265] := 16#A5E1;
   // UNICODE_TO_GBK[1266] := 16#30E2;
   // UNICODE_TO_GBK[1267] := 16#A5E2;
   // UNICODE_TO_GBK[1268] := 16#30E3;
   // UNICODE_TO_GBK[1269] := 16#A5E3;
   // UNICODE_TO_GBK[1270] := 16#30E4;
   // UNICODE_TO_GBK[1271] := 16#A5E4;
   // UNICODE_TO_GBK[1272] := 16#30E5;
   // UNICODE_TO_GBK[1273] := 16#A5E5;
   // UNICODE_TO_GBK[1274] := 16#30E6;
   // UNICODE_TO_GBK[1275] := 16#A5E6;
   // UNICODE_TO_GBK[1276] := 16#30E7;
   // UNICODE_TO_GBK[1277] := 16#A5E7;
   // UNICODE_TO_GBK[1278] := 16#30E8;
   // UNICODE_TO_GBK[1279] := 16#A5E8;
   // UNICODE_TO_GBK[1280] := 16#30E9;
   // UNICODE_TO_GBK[1281] := 16#A5E9;
   // UNICODE_TO_GBK[1282] := 16#30EA;
   // UNICODE_TO_GBK[1283] := 16#A5EA;
   // UNICODE_TO_GBK[1284] := 16#30EB;
   // UNICODE_TO_GBK[1285] := 16#A5EB;
   // UNICODE_TO_GBK[1286] := 16#30EC;
   // UNICODE_TO_GBK[1287] := 16#A5EC;
   // UNICODE_TO_GBK[1288] := 16#30ED;
   // UNICODE_TO_GBK[1289] := 16#A5ED;
   // UNICODE_TO_GBK[1290] := 16#30EE;
   // UNICODE_TO_GBK[1291] := 16#A5EE;
   // UNICODE_TO_GBK[1292] := 16#30EF;
   // UNICODE_TO_GBK[1293] := 16#A5EF;
   // UNICODE_TO_GBK[1294] := 16#30F0;
   // UNICODE_TO_GBK[1295] := 16#A5F0;
   // UNICODE_TO_GBK[1296] := 16#30F1;
   // UNICODE_TO_GBK[1297] := 16#A5F1;
   // UNICODE_TO_GBK[1298] := 16#30F2;
   // UNICODE_TO_GBK[1299] := 16#A5F2;
   // UNICODE_TO_GBK[1300] := 16#30F3;
   // UNICODE_TO_GBK[1301] := 16#A5F3;
   // UNICODE_TO_GBK[1302] := 16#30F4;
   // UNICODE_TO_GBK[1303] := 16#A5F4;
   // UNICODE_TO_GBK[1304] := 16#30F5;
   // UNICODE_TO_GBK[1305] := 16#A5F5;
   // UNICODE_TO_GBK[1306] := 16#30F6;
   // UNICODE_TO_GBK[1307] := 16#A5F6;
   // UNICODE_TO_GBK[1308] := 16#30FC;
   // UNICODE_TO_GBK[1309] := 16#A960;
   // UNICODE_TO_GBK[1310] := 16#30FD;
   // UNICODE_TO_GBK[1311] := 16#A963;
   // UNICODE_TO_GBK[1312] := 16#30FE;
   // UNICODE_TO_GBK[1313] := 16#A964;
   // UNICODE_TO_GBK[1314] := 16#3105;
   // UNICODE_TO_GBK[1315] := 16#A8C5;
   // UNICODE_TO_GBK[1316] := 16#3106;
   // UNICODE_TO_GBK[1317] := 16#A8C6;
   // UNICODE_TO_GBK[1318] := 16#3107;
   // UNICODE_TO_GBK[1319] := 16#A8C7;
   // UNICODE_TO_GBK[1320] := 16#3108;
   // UNICODE_TO_GBK[1321] := 16#A8C8;
   // UNICODE_TO_GBK[1322] := 16#3109;
   // UNICODE_TO_GBK[1323] := 16#A8C9;
   // UNICODE_TO_GBK[1324] := 16#310A;
   // UNICODE_TO_GBK[1325] := 16#A8CA;
   // UNICODE_TO_GBK[1326] := 16#310B;
   // UNICODE_TO_GBK[1327] := 16#A8CB;
   // UNICODE_TO_GBK[1328] := 16#310C;
   // UNICODE_TO_GBK[1329] := 16#A8CC;
   // UNICODE_TO_GBK[1330] := 16#310D;
   // UNICODE_TO_GBK[1331] := 16#A8CD;
   // UNICODE_TO_GBK[1332] := 16#310E;
   // UNICODE_TO_GBK[1333] := 16#A8CE;
   // UNICODE_TO_GBK[1334] := 16#310F;
   // UNICODE_TO_GBK[1335] := 16#A8CF;
   // UNICODE_TO_GBK[1336] := 16#3110;
   // UNICODE_TO_GBK[1337] := 16#A8D0;
   // UNICODE_TO_GBK[1338] := 16#3111;
   // UNICODE_TO_GBK[1339] := 16#A8D1;
   // UNICODE_TO_GBK[1340] := 16#3112;
   // UNICODE_TO_GBK[1341] := 16#A8D2;
   // UNICODE_TO_GBK[1342] := 16#3113;
   // UNICODE_TO_GBK[1343] := 16#A8D3;
   // UNICODE_TO_GBK[1344] := 16#3114;
   // UNICODE_TO_GBK[1345] := 16#A8D4;
   // UNICODE_TO_GBK[1346] := 16#3115;
   // UNICODE_TO_GBK[1347] := 16#A8D5;
   // UNICODE_TO_GBK[1348] := 16#3116;
   // UNICODE_TO_GBK[1349] := 16#A8D6;
   // UNICODE_TO_GBK[1350] := 16#3117;
   // UNICODE_TO_GBK[1351] := 16#A8D7;
   // UNICODE_TO_GBK[1352] := 16#3118;
   // UNICODE_TO_GBK[1353] := 16#A8D8;
   // UNICODE_TO_GBK[1354] := 16#3119;
   // UNICODE_TO_GBK[1355] := 16#A8D9;
   // UNICODE_TO_GBK[1356] := 16#311A;
   // UNICODE_TO_GBK[1357] := 16#A8DA;
   // UNICODE_TO_GBK[1358] := 16#311B;
   // UNICODE_TO_GBK[1359] := 16#A8DB;
   // UNICODE_TO_GBK[1360] := 16#311C;
   // UNICODE_TO_GBK[1361] := 16#A8DC;
   // UNICODE_TO_GBK[1362] := 16#311D;
   // UNICODE_TO_GBK[1363] := 16#A8DD;
   // UNICODE_TO_GBK[1364] := 16#311E;
   // UNICODE_TO_GBK[1365] := 16#A8DE;
   // UNICODE_TO_GBK[1366] := 16#311F;
   // UNICODE_TO_GBK[1367] := 16#A8DF;
   // UNICODE_TO_GBK[1368] := 16#3120;
   // UNICODE_TO_GBK[1369] := 16#A8E0;
   // UNICODE_TO_GBK[1370] := 16#3121;
   // UNICODE_TO_GBK[1371] := 16#A8E1;
   // UNICODE_TO_GBK[1372] := 16#3122;
   // UNICODE_TO_GBK[1373] := 16#A8E2;
   // UNICODE_TO_GBK[1374] := 16#3123;
   // UNICODE_TO_GBK[1375] := 16#A8E3;
   // UNICODE_TO_GBK[1376] := 16#3124;
   // UNICODE_TO_GBK[1377] := 16#A8E4;
   // UNICODE_TO_GBK[1378] := 16#3125;
   // UNICODE_TO_GBK[1379] := 16#A8E5;
   // UNICODE_TO_GBK[1380] := 16#3126;
   // UNICODE_TO_GBK[1381] := 16#A8E6;
   // UNICODE_TO_GBK[1382] := 16#3127;
   // UNICODE_TO_GBK[1383] := 16#A8E7;
   // UNICODE_TO_GBK[1384] := 16#3128;
   // UNICODE_TO_GBK[1385] := 16#A8E8;
   // UNICODE_TO_GBK[1386] := 16#3129;
   // UNICODE_TO_GBK[1387] := 16#A8E9;
   // UNICODE_TO_GBK[1388] := 16#3220;
   // UNICODE_TO_GBK[1389] := 16#A2E5;
   // UNICODE_TO_GBK[1390] := 16#3221;
   // UNICODE_TO_GBK[1391] := 16#A2E6;
   // UNICODE_TO_GBK[1392] := 16#3222;
   // UNICODE_TO_GBK[1393] := 16#A2E7;
   // UNICODE_TO_GBK[1394] := 16#3223;
   // UNICODE_TO_GBK[1395] := 16#A2E8;
   // UNICODE_TO_GBK[1396] := 16#3224;
   // UNICODE_TO_GBK[1397] := 16#A2E9;
   // UNICODE_TO_GBK[1398] := 16#3225;
   // UNICODE_TO_GBK[1399] := 16#A2EA;
   // UNICODE_TO_GBK[1400] := 16#3226;
   // UNICODE_TO_GBK[1401] := 16#A2EB;
   // UNICODE_TO_GBK[1402] := 16#3227;
   // UNICODE_TO_GBK[1403] := 16#A2EC;
   // UNICODE_TO_GBK[1404] := 16#3228;
   // UNICODE_TO_GBK[1405] := 16#A2ED;
   // UNICODE_TO_GBK[1406] := 16#3229;
   // UNICODE_TO_GBK[1407] := 16#A2EE;
   // UNICODE_TO_GBK[1408] := 16#3231;
   // UNICODE_TO_GBK[1409] := 16#A95A;
   // UNICODE_TO_GBK[1410] := 16#32A3;
   // UNICODE_TO_GBK[1411] := 16#A949;
   // UNICODE_TO_GBK[1412] := 16#338E;
   // UNICODE_TO_GBK[1413] := 16#A94A;
   // UNICODE_TO_GBK[1414] := 16#338F;
   // UNICODE_TO_GBK[1415] := 16#A94B;
   // UNICODE_TO_GBK[1416] := 16#339C;
   // UNICODE_TO_GBK[1417] := 16#A94C;
   // UNICODE_TO_GBK[1418] := 16#339D;
   // UNICODE_TO_GBK[1419] := 16#A94D;
   // UNICODE_TO_GBK[1420] := 16#339E;
   // UNICODE_TO_GBK[1421] := 16#A94E;
   // UNICODE_TO_GBK[1422] := 16#33A1;
   // UNICODE_TO_GBK[1423] := 16#A94F;
   // UNICODE_TO_GBK[1424] := 16#33C4;
   // UNICODE_TO_GBK[1425] := 16#A950;
   // UNICODE_TO_GBK[1426] := 16#33CE;
   // UNICODE_TO_GBK[1427] := 16#A951;
   // UNICODE_TO_GBK[1428] := 16#33D1;
   // UNICODE_TO_GBK[1429] := 16#A952;
   // UNICODE_TO_GBK[1430] := 16#33D2;
   // UNICODE_TO_GBK[1431] := 16#A953;
   // UNICODE_TO_GBK[1432] := 16#33D5;
   // UNICODE_TO_GBK[1433] := 16#A954;
   // UNICODE_TO_GBK[1434] := 16#4E00;
   // UNICODE_TO_GBK[1435] := 16#D2BB;
   // UNICODE_TO_GBK[1436] := 16#4E01;
   // UNICODE_TO_GBK[1437] := 16#B6A1;
   // UNICODE_TO_GBK[1438] := 16#4E02;
   // UNICODE_TO_GBK[1439] := 16#8140;
   // UNICODE_TO_GBK[1440] := 16#4E03;
   // UNICODE_TO_GBK[1441] := 16#C6DF;
   // UNICODE_TO_GBK[1442] := 16#4E04;
   // UNICODE_TO_GBK[1443] := 16#8141;
   // UNICODE_TO_GBK[1444] := 16#4E05;
   // UNICODE_TO_GBK[1445] := 16#8142;
   // UNICODE_TO_GBK[1446] := 16#4E06;
   // UNICODE_TO_GBK[1447] := 16#8143;
   // UNICODE_TO_GBK[1448] := 16#4E07;
   // UNICODE_TO_GBK[1449] := 16#CDF2;
   // UNICODE_TO_GBK[1450] := 16#4E08;
   // UNICODE_TO_GBK[1451] := 16#D5C9;
   // UNICODE_TO_GBK[1452] := 16#4E09;
   // UNICODE_TO_GBK[1453] := 16#C8FD;
   // UNICODE_TO_GBK[1454] := 16#4E0A;
   // UNICODE_TO_GBK[1455] := 16#C9CF;
   // UNICODE_TO_GBK[1456] := 16#4E0B;
   // UNICODE_TO_GBK[1457] := 16#CFC2;
   // UNICODE_TO_GBK[1458] := 16#4E0C;
   // UNICODE_TO_GBK[1459] := 16#D8A2;
   // UNICODE_TO_GBK[1460] := 16#4E0D;
   // UNICODE_TO_GBK[1461] := 16#B2BB;
   // UNICODE_TO_GBK[1462] := 16#4E0E;
   // UNICODE_TO_GBK[1463] := 16#D3EB;
   // UNICODE_TO_GBK[1464] := 16#4E0F;
   // UNICODE_TO_GBK[1465] := 16#8144;
   // UNICODE_TO_GBK[1466] := 16#4E10;
   // UNICODE_TO_GBK[1467] := 16#D8A4;
   // UNICODE_TO_GBK[1468] := 16#4E11;
   // UNICODE_TO_GBK[1469] := 16#B3F3;
   // UNICODE_TO_GBK[1470] := 16#4E12;
   // UNICODE_TO_GBK[1471] := 16#8145;
   // UNICODE_TO_GBK[1472] := 16#4E13;
   // UNICODE_TO_GBK[1473] := 16#D7A8;
   // UNICODE_TO_GBK[1474] := 16#4E14;
   // UNICODE_TO_GBK[1475] := 16#C7D2;
   // UNICODE_TO_GBK[1476] := 16#4E15;
   // UNICODE_TO_GBK[1477] := 16#D8A7;
   // UNICODE_TO_GBK[1478] := 16#4E16;
   // UNICODE_TO_GBK[1479] := 16#CAC0;
   // UNICODE_TO_GBK[1480] := 16#4E17;
   // UNICODE_TO_GBK[1481] := 16#8146;
   // UNICODE_TO_GBK[1482] := 16#4E18;
   // UNICODE_TO_GBK[1483] := 16#C7F0;
   // UNICODE_TO_GBK[1484] := 16#4E19;
   // UNICODE_TO_GBK[1485] := 16#B1FB;
   // UNICODE_TO_GBK[1486] := 16#4E1A;
   // UNICODE_TO_GBK[1487] := 16#D2B5;
   // UNICODE_TO_GBK[1488] := 16#4E1B;
   // UNICODE_TO_GBK[1489] := 16#B4D4;
   // UNICODE_TO_GBK[1490] := 16#4E1C;
   // UNICODE_TO_GBK[1491] := 16#B6AB;
   // UNICODE_TO_GBK[1492] := 16#4E1D;
   // UNICODE_TO_GBK[1493] := 16#CBBF;
   // UNICODE_TO_GBK[1494] := 16#4E1E;
   // UNICODE_TO_GBK[1495] := 16#D8A9;
   // UNICODE_TO_GBK[1496] := 16#4E1F;
   // UNICODE_TO_GBK[1497] := 16#8147;
   // UNICODE_TO_GBK[1498] := 16#4E20;
   // UNICODE_TO_GBK[1499] := 16#8148;
   // UNICODE_TO_GBK[1500] := 16#4E21;
   // UNICODE_TO_GBK[1501] := 16#8149;
   // UNICODE_TO_GBK[1502] := 16#4E22;
   // UNICODE_TO_GBK[1503] := 16#B6AA;
   // UNICODE_TO_GBK[1504] := 16#4E23;
   // UNICODE_TO_GBK[1505] := 16#814A;
   // UNICODE_TO_GBK[1506] := 16#4E24;
   // UNICODE_TO_GBK[1507] := 16#C1BD;
   // UNICODE_TO_GBK[1508] := 16#4E25;
   // UNICODE_TO_GBK[1509] := 16#D1CF;
   // UNICODE_TO_GBK[1510] := 16#4E26;
   // UNICODE_TO_GBK[1511] := 16#814B;
   // UNICODE_TO_GBK[1512] := 16#4E27;
   // UNICODE_TO_GBK[1513] := 16#C9A5;
   // UNICODE_TO_GBK[1514] := 16#4E28;
   // UNICODE_TO_GBK[1515] := 16#D8AD;
   // UNICODE_TO_GBK[1516] := 16#4E29;
   // UNICODE_TO_GBK[1517] := 16#814C;
   // UNICODE_TO_GBK[1518] := 16#4E2A;
   // UNICODE_TO_GBK[1519] := 16#B8F6;
   // UNICODE_TO_GBK[1520] := 16#4E2B;
   // UNICODE_TO_GBK[1521] := 16#D1BE;
   // UNICODE_TO_GBK[1522] := 16#4E2C;
   // UNICODE_TO_GBK[1523] := 16#E3DC;
   // UNICODE_TO_GBK[1524] := 16#4E2D;
   // UNICODE_TO_GBK[1525] := 16#D6D0;
   // UNICODE_TO_GBK[1526] := 16#4E2E;
   // UNICODE_TO_GBK[1527] := 16#814D;
   // UNICODE_TO_GBK[1528] := 16#4E2F;
   // UNICODE_TO_GBK[1529] := 16#814E;
   // UNICODE_TO_GBK[1530] := 16#4E30;
   // UNICODE_TO_GBK[1531] := 16#B7E1;
   // UNICODE_TO_GBK[1532] := 16#4E31;
   // UNICODE_TO_GBK[1533] := 16#814F;
   // UNICODE_TO_GBK[1534] := 16#4E32;
   // UNICODE_TO_GBK[1535] := 16#B4AE;
   // UNICODE_TO_GBK[1536] := 16#4E33;
   // UNICODE_TO_GBK[1537] := 16#8150;
   // UNICODE_TO_GBK[1538] := 16#4E34;
   // UNICODE_TO_GBK[1539] := 16#C1D9;
   // UNICODE_TO_GBK[1540] := 16#4E35;
   // UNICODE_TO_GBK[1541] := 16#8151;
   // UNICODE_TO_GBK[1542] := 16#4E36;
   // UNICODE_TO_GBK[1543] := 16#D8BC;
   // UNICODE_TO_GBK[1544] := 16#4E37;
   // UNICODE_TO_GBK[1545] := 16#8152;
   // UNICODE_TO_GBK[1546] := 16#4E38;
   // UNICODE_TO_GBK[1547] := 16#CDE8;
   // UNICODE_TO_GBK[1548] := 16#4E39;
   // UNICODE_TO_GBK[1549] := 16#B5A4;
   // UNICODE_TO_GBK[1550] := 16#4E3A;
   // UNICODE_TO_GBK[1551] := 16#CEAA;
   // UNICODE_TO_GBK[1552] := 16#4E3B;
   // UNICODE_TO_GBK[1553] := 16#D6F7;
   // UNICODE_TO_GBK[1554] := 16#4E3C;
   // UNICODE_TO_GBK[1555] := 16#8153;
   // UNICODE_TO_GBK[1556] := 16#4E3D;
   // UNICODE_TO_GBK[1557] := 16#C0F6;
   // UNICODE_TO_GBK[1558] := 16#4E3E;
   // UNICODE_TO_GBK[1559] := 16#BED9;
   // UNICODE_TO_GBK[1560] := 16#4E3F;
   // UNICODE_TO_GBK[1561] := 16#D8AF;
   // UNICODE_TO_GBK[1562] := 16#4E40;
   // UNICODE_TO_GBK[1563] := 16#8154;
   // UNICODE_TO_GBK[1564] := 16#4E41;
   // UNICODE_TO_GBK[1565] := 16#8155;
   // UNICODE_TO_GBK[1566] := 16#4E42;
   // UNICODE_TO_GBK[1567] := 16#8156;
   // UNICODE_TO_GBK[1568] := 16#4E43;
   // UNICODE_TO_GBK[1569] := 16#C4CB;
   // UNICODE_TO_GBK[1570] := 16#4E44;
   // UNICODE_TO_GBK[1571] := 16#8157;
   // UNICODE_TO_GBK[1572] := 16#4E45;
   // UNICODE_TO_GBK[1573] := 16#BEC3;
   // UNICODE_TO_GBK[1574] := 16#4E46;
   // UNICODE_TO_GBK[1575] := 16#8158;
   // UNICODE_TO_GBK[1576] := 16#4E47;
   // UNICODE_TO_GBK[1577] := 16#D8B1;
   // UNICODE_TO_GBK[1578] := 16#4E48;
   // UNICODE_TO_GBK[1579] := 16#C3B4;
   // UNICODE_TO_GBK[1580] := 16#4E49;
   // UNICODE_TO_GBK[1581] := 16#D2E5;
   // UNICODE_TO_GBK[1582] := 16#4E4A;
   // UNICODE_TO_GBK[1583] := 16#8159;
   // UNICODE_TO_GBK[1584] := 16#4E4B;
   // UNICODE_TO_GBK[1585] := 16#D6AE;
   // UNICODE_TO_GBK[1586] := 16#4E4C;
   // UNICODE_TO_GBK[1587] := 16#CEDA;
   // UNICODE_TO_GBK[1588] := 16#4E4D;
   // UNICODE_TO_GBK[1589] := 16#D5A7;
   // UNICODE_TO_GBK[1590] := 16#4E4E;
   // UNICODE_TO_GBK[1591] := 16#BAF5;
   // UNICODE_TO_GBK[1592] := 16#4E4F;
   // UNICODE_TO_GBK[1593] := 16#B7A6;
   // UNICODE_TO_GBK[1594] := 16#4E50;
   // UNICODE_TO_GBK[1595] := 16#C0D6;
   // UNICODE_TO_GBK[1596] := 16#4E51;
   // UNICODE_TO_GBK[1597] := 16#815A;
   // UNICODE_TO_GBK[1598] := 16#4E52;
   // UNICODE_TO_GBK[1599] := 16#C6B9;
   // UNICODE_TO_GBK[1600] := 16#4E53;
   // UNICODE_TO_GBK[1601] := 16#C5D2;
   // UNICODE_TO_GBK[1602] := 16#4E54;
   // UNICODE_TO_GBK[1603] := 16#C7C7;
   // UNICODE_TO_GBK[1604] := 16#4E55;
   // UNICODE_TO_GBK[1605] := 16#815B;
   // UNICODE_TO_GBK[1606] := 16#4E56;
   // UNICODE_TO_GBK[1607] := 16#B9D4;
   // UNICODE_TO_GBK[1608] := 16#4E57;
   // UNICODE_TO_GBK[1609] := 16#815C;
   // UNICODE_TO_GBK[1610] := 16#4E58;
   // UNICODE_TO_GBK[1611] := 16#B3CB;
   // UNICODE_TO_GBK[1612] := 16#4E59;
   // UNICODE_TO_GBK[1613] := 16#D2D2;
   // UNICODE_TO_GBK[1614] := 16#4E5A;
   // UNICODE_TO_GBK[1615] := 16#815D;
   // UNICODE_TO_GBK[1616] := 16#4E5B;
   // UNICODE_TO_GBK[1617] := 16#815E;
   // UNICODE_TO_GBK[1618] := 16#4E5C;
   // UNICODE_TO_GBK[1619] := 16#D8BF;
   // UNICODE_TO_GBK[1620] := 16#4E5D;
   // UNICODE_TO_GBK[1621] := 16#BEC5;
   // UNICODE_TO_GBK[1622] := 16#4E5E;
   // UNICODE_TO_GBK[1623] := 16#C6F2;
   // UNICODE_TO_GBK[1624] := 16#4E5F;
   // UNICODE_TO_GBK[1625] := 16#D2B2;
   // UNICODE_TO_GBK[1626] := 16#4E60;
   // UNICODE_TO_GBK[1627] := 16#CFB0;
   // UNICODE_TO_GBK[1628] := 16#4E61;
   // UNICODE_TO_GBK[1629] := 16#CFE7;
   // UNICODE_TO_GBK[1630] := 16#4E62;
   // UNICODE_TO_GBK[1631] := 16#815F;
   // UNICODE_TO_GBK[1632] := 16#4E63;
   // UNICODE_TO_GBK[1633] := 16#8160;
   // UNICODE_TO_GBK[1634] := 16#4E64;
   // UNICODE_TO_GBK[1635] := 16#8161;
   // UNICODE_TO_GBK[1636] := 16#4E65;
   // UNICODE_TO_GBK[1637] := 16#8162;
   // UNICODE_TO_GBK[1638] := 16#4E66;
   // UNICODE_TO_GBK[1639] := 16#CAE9;
   // UNICODE_TO_GBK[1640] := 16#4E67;
   // UNICODE_TO_GBK[1641] := 16#8163;
   // UNICODE_TO_GBK[1642] := 16#4E68;
   // UNICODE_TO_GBK[1643] := 16#8164;
   // UNICODE_TO_GBK[1644] := 16#4E69;
   // UNICODE_TO_GBK[1645] := 16#D8C0;
   // UNICODE_TO_GBK[1646] := 16#4E6A;
   // UNICODE_TO_GBK[1647] := 16#8165;
   // UNICODE_TO_GBK[1648] := 16#4E6B;
   // UNICODE_TO_GBK[1649] := 16#8166;
   // UNICODE_TO_GBK[1650] := 16#4E6C;
   // UNICODE_TO_GBK[1651] := 16#8167;
   // UNICODE_TO_GBK[1652] := 16#4E6D;
   // UNICODE_TO_GBK[1653] := 16#8168;
   // UNICODE_TO_GBK[1654] := 16#4E6E;
   // UNICODE_TO_GBK[1655] := 16#8169;
   // UNICODE_TO_GBK[1656] := 16#4E6F;
   // UNICODE_TO_GBK[1657] := 16#816A;
   // UNICODE_TO_GBK[1658] := 16#4E70;
   // UNICODE_TO_GBK[1659] := 16#C2F2;
   // UNICODE_TO_GBK[1660] := 16#4E71;
   // UNICODE_TO_GBK[1661] := 16#C2D2;
   // UNICODE_TO_GBK[1662] := 16#4E72;
   // UNICODE_TO_GBK[1663] := 16#816B;
   // UNICODE_TO_GBK[1664] := 16#4E73;
   // UNICODE_TO_GBK[1665] := 16#C8E9;
   // UNICODE_TO_GBK[1666] := 16#4E74;
   // UNICODE_TO_GBK[1667] := 16#816C;
   // UNICODE_TO_GBK[1668] := 16#4E75;
   // UNICODE_TO_GBK[1669] := 16#816D;
   // UNICODE_TO_GBK[1670] := 16#4E76;
   // UNICODE_TO_GBK[1671] := 16#816E;
   // UNICODE_TO_GBK[1672] := 16#4E77;
   // UNICODE_TO_GBK[1673] := 16#816F;
   // UNICODE_TO_GBK[1674] := 16#4E78;
   // UNICODE_TO_GBK[1675] := 16#8170;
   // UNICODE_TO_GBK[1676] := 16#4E79;
   // UNICODE_TO_GBK[1677] := 16#8171;
   // UNICODE_TO_GBK[1678] := 16#4E7A;
   // UNICODE_TO_GBK[1679] := 16#8172;
   // UNICODE_TO_GBK[1680] := 16#4E7B;
   // UNICODE_TO_GBK[1681] := 16#8173;
   // UNICODE_TO_GBK[1682] := 16#4E7C;
   // UNICODE_TO_GBK[1683] := 16#8174;
   // UNICODE_TO_GBK[1684] := 16#4E7D;
   // UNICODE_TO_GBK[1685] := 16#8175;
   // UNICODE_TO_GBK[1686] := 16#4E7E;
   // UNICODE_TO_GBK[1687] := 16#C7AC;
   // UNICODE_TO_GBK[1688] := 16#4E7F;
   // UNICODE_TO_GBK[1689] := 16#8176;
   // UNICODE_TO_GBK[1690] := 16#4E80;
   // UNICODE_TO_GBK[1691] := 16#8177;
   // UNICODE_TO_GBK[1692] := 16#4E81;
   // UNICODE_TO_GBK[1693] := 16#8178;
   // UNICODE_TO_GBK[1694] := 16#4E82;
   // UNICODE_TO_GBK[1695] := 16#8179;
   // UNICODE_TO_GBK[1696] := 16#4E83;
   // UNICODE_TO_GBK[1697] := 16#817A;
   // UNICODE_TO_GBK[1698] := 16#4E84;
   // UNICODE_TO_GBK[1699] := 16#817B;
   // UNICODE_TO_GBK[1700] := 16#4E85;
   // UNICODE_TO_GBK[1701] := 16#817C;
   // UNICODE_TO_GBK[1702] := 16#4E86;
   // UNICODE_TO_GBK[1703] := 16#C1CB;
   // UNICODE_TO_GBK[1704] := 16#4E87;
   // UNICODE_TO_GBK[1705] := 16#817D;
   // UNICODE_TO_GBK[1706] := 16#4E88;
   // UNICODE_TO_GBK[1707] := 16#D3E8;
   // UNICODE_TO_GBK[1708] := 16#4E89;
   // UNICODE_TO_GBK[1709] := 16#D5F9;
   // UNICODE_TO_GBK[1710] := 16#4E8A;
   // UNICODE_TO_GBK[1711] := 16#817E;
   // UNICODE_TO_GBK[1712] := 16#4E8B;
   // UNICODE_TO_GBK[1713] := 16#CAC2;
   // UNICODE_TO_GBK[1714] := 16#4E8C;
   // UNICODE_TO_GBK[1715] := 16#B6FE;
   // UNICODE_TO_GBK[1716] := 16#4E8D;
   // UNICODE_TO_GBK[1717] := 16#D8A1;
   // UNICODE_TO_GBK[1718] := 16#4E8E;
   // UNICODE_TO_GBK[1719] := 16#D3DA;
   // UNICODE_TO_GBK[1720] := 16#4E8F;
   // UNICODE_TO_GBK[1721] := 16#BFF7;
   // UNICODE_TO_GBK[1722] := 16#4E90;
   // UNICODE_TO_GBK[1723] := 16#8180;
   // UNICODE_TO_GBK[1724] := 16#4E91;
   // UNICODE_TO_GBK[1725] := 16#D4C6;
   // UNICODE_TO_GBK[1726] := 16#4E92;
   // UNICODE_TO_GBK[1727] := 16#BBA5;
   // UNICODE_TO_GBK[1728] := 16#4E93;
   // UNICODE_TO_GBK[1729] := 16#D8C1;
   // UNICODE_TO_GBK[1730] := 16#4E94;
   // UNICODE_TO_GBK[1731] := 16#CEE5;
   // UNICODE_TO_GBK[1732] := 16#4E95;
   // UNICODE_TO_GBK[1733] := 16#BEAE;
   // UNICODE_TO_GBK[1734] := 16#4E96;
   // UNICODE_TO_GBK[1735] := 16#8181;
   // UNICODE_TO_GBK[1736] := 16#4E97;
   // UNICODE_TO_GBK[1737] := 16#8182;
   // UNICODE_TO_GBK[1738] := 16#4E98;
   // UNICODE_TO_GBK[1739] := 16#D8A8;
   // UNICODE_TO_GBK[1740] := 16#4E99;
   // UNICODE_TO_GBK[1741] := 16#8183;
   // UNICODE_TO_GBK[1742] := 16#4E9A;
   // UNICODE_TO_GBK[1743] := 16#D1C7;
   // UNICODE_TO_GBK[1744] := 16#4E9B;
   // UNICODE_TO_GBK[1745] := 16#D0A9;
   // UNICODE_TO_GBK[1746] := 16#4E9C;
   // UNICODE_TO_GBK[1747] := 16#8184;
   // UNICODE_TO_GBK[1748] := 16#4E9D;
   // UNICODE_TO_GBK[1749] := 16#8185;
   // UNICODE_TO_GBK[1750] := 16#4E9E;
   // UNICODE_TO_GBK[1751] := 16#8186;
   // UNICODE_TO_GBK[1752] := 16#4E9F;
   // UNICODE_TO_GBK[1753] := 16#D8BD;
   // UNICODE_TO_GBK[1754] := 16#4EA0;
   // UNICODE_TO_GBK[1755] := 16#D9EF;
   // UNICODE_TO_GBK[1756] := 16#4EA1;
   // UNICODE_TO_GBK[1757] := 16#CDF6;
   // UNICODE_TO_GBK[1758] := 16#4EA2;
   // UNICODE_TO_GBK[1759] := 16#BFBA;
   // UNICODE_TO_GBK[1760] := 16#4EA3;
   // UNICODE_TO_GBK[1761] := 16#8187;
   // UNICODE_TO_GBK[1762] := 16#4EA4;
   // UNICODE_TO_GBK[1763] := 16#BDBB;
   // UNICODE_TO_GBK[1764] := 16#4EA5;
   // UNICODE_TO_GBK[1765] := 16#BAA5;
   // UNICODE_TO_GBK[1766] := 16#4EA6;
   // UNICODE_TO_GBK[1767] := 16#D2E0;
   // UNICODE_TO_GBK[1768] := 16#4EA7;
   // UNICODE_TO_GBK[1769] := 16#B2FA;
   // UNICODE_TO_GBK[1770] := 16#4EA8;
   // UNICODE_TO_GBK[1771] := 16#BAE0;
   // UNICODE_TO_GBK[1772] := 16#4EA9;
   // UNICODE_TO_GBK[1773] := 16#C4B6;
   // UNICODE_TO_GBK[1774] := 16#4EAA;
   // UNICODE_TO_GBK[1775] := 16#8188;
   // UNICODE_TO_GBK[1776] := 16#4EAB;
   // UNICODE_TO_GBK[1777] := 16#CFED;
   // UNICODE_TO_GBK[1778] := 16#4EAC;
   // UNICODE_TO_GBK[1779] := 16#BEA9;
   // UNICODE_TO_GBK[1780] := 16#4EAD;
   // UNICODE_TO_GBK[1781] := 16#CDA4;
   // UNICODE_TO_GBK[1782] := 16#4EAE;
   // UNICODE_TO_GBK[1783] := 16#C1C1;
   // UNICODE_TO_GBK[1784] := 16#4EAF;
   // UNICODE_TO_GBK[1785] := 16#8189;
   // UNICODE_TO_GBK[1786] := 16#4EB0;
   // UNICODE_TO_GBK[1787] := 16#818A;
   // UNICODE_TO_GBK[1788] := 16#4EB1;
   // UNICODE_TO_GBK[1789] := 16#818B;
   // UNICODE_TO_GBK[1790] := 16#4EB2;
   // UNICODE_TO_GBK[1791] := 16#C7D7;
   // UNICODE_TO_GBK[1792] := 16#4EB3;
   // UNICODE_TO_GBK[1793] := 16#D9F1;
   // UNICODE_TO_GBK[1794] := 16#4EB4;
   // UNICODE_TO_GBK[1795] := 16#818C;
   // UNICODE_TO_GBK[1796] := 16#4EB5;
   // UNICODE_TO_GBK[1797] := 16#D9F4;
   // UNICODE_TO_GBK[1798] := 16#4EB6;
   // UNICODE_TO_GBK[1799] := 16#818D;
   // UNICODE_TO_GBK[1800] := 16#4EB7;
   // UNICODE_TO_GBK[1801] := 16#818E;
   // UNICODE_TO_GBK[1802] := 16#4EB8;
   // UNICODE_TO_GBK[1803] := 16#818F;
   // UNICODE_TO_GBK[1804] := 16#4EB9;
   // UNICODE_TO_GBK[1805] := 16#8190;
   // UNICODE_TO_GBK[1806] := 16#4EBA;
   // UNICODE_TO_GBK[1807] := 16#C8CB;
   // UNICODE_TO_GBK[1808] := 16#4EBB;
   // UNICODE_TO_GBK[1809] := 16#D8E9;
   // UNICODE_TO_GBK[1810] := 16#4EBC;
   // UNICODE_TO_GBK[1811] := 16#8191;
   // UNICODE_TO_GBK[1812] := 16#4EBD;
   // UNICODE_TO_GBK[1813] := 16#8192;
   // UNICODE_TO_GBK[1814] := 16#4EBE;
   // UNICODE_TO_GBK[1815] := 16#8193;
   // UNICODE_TO_GBK[1816] := 16#4EBF;
   // UNICODE_TO_GBK[1817] := 16#D2DA;
   // UNICODE_TO_GBK[1818] := 16#4EC0;
   // UNICODE_TO_GBK[1819] := 16#CAB2;
   // UNICODE_TO_GBK[1820] := 16#4EC1;
   // UNICODE_TO_GBK[1821] := 16#C8CA;
   // UNICODE_TO_GBK[1822] := 16#4EC2;
   // UNICODE_TO_GBK[1823] := 16#D8EC;
   // UNICODE_TO_GBK[1824] := 16#4EC3;
   // UNICODE_TO_GBK[1825] := 16#D8EA;
   // UNICODE_TO_GBK[1826] := 16#4EC4;
   // UNICODE_TO_GBK[1827] := 16#D8C6;
   // UNICODE_TO_GBK[1828] := 16#4EC5;
   // UNICODE_TO_GBK[1829] := 16#BDF6;
   // UNICODE_TO_GBK[1830] := 16#4EC6;
   // UNICODE_TO_GBK[1831] := 16#C6CD;
   // UNICODE_TO_GBK[1832] := 16#4EC7;
   // UNICODE_TO_GBK[1833] := 16#B3F0;
   // UNICODE_TO_GBK[1834] := 16#4EC8;
   // UNICODE_TO_GBK[1835] := 16#8194;
   // UNICODE_TO_GBK[1836] := 16#4EC9;
   // UNICODE_TO_GBK[1837] := 16#D8EB;
   // UNICODE_TO_GBK[1838] := 16#4ECA;
   // UNICODE_TO_GBK[1839] := 16#BDF1;
   // UNICODE_TO_GBK[1840] := 16#4ECB;
   // UNICODE_TO_GBK[1841] := 16#BDE9;
   // UNICODE_TO_GBK[1842] := 16#4ECC;
   // UNICODE_TO_GBK[1843] := 16#8195;
   // UNICODE_TO_GBK[1844] := 16#4ECD;
   // UNICODE_TO_GBK[1845] := 16#C8D4;
   // UNICODE_TO_GBK[1846] := 16#4ECE;
   // UNICODE_TO_GBK[1847] := 16#B4D3;
   // UNICODE_TO_GBK[1848] := 16#4ECF;
   // UNICODE_TO_GBK[1849] := 16#8196;
   // UNICODE_TO_GBK[1850] := 16#4ED0;
   // UNICODE_TO_GBK[1851] := 16#8197;
   // UNICODE_TO_GBK[1852] := 16#4ED1;
   // UNICODE_TO_GBK[1853] := 16#C2D8;
   // UNICODE_TO_GBK[1854] := 16#4ED2;
   // UNICODE_TO_GBK[1855] := 16#8198;
   // UNICODE_TO_GBK[1856] := 16#4ED3;
   // UNICODE_TO_GBK[1857] := 16#B2D6;
   // UNICODE_TO_GBK[1858] := 16#4ED4;
   // UNICODE_TO_GBK[1859] := 16#D7D0;
   // UNICODE_TO_GBK[1860] := 16#4ED5;
   // UNICODE_TO_GBK[1861] := 16#CACB;
   // UNICODE_TO_GBK[1862] := 16#4ED6;
   // UNICODE_TO_GBK[1863] := 16#CBFB;
   // UNICODE_TO_GBK[1864] := 16#4ED7;
   // UNICODE_TO_GBK[1865] := 16#D5CC;
   // UNICODE_TO_GBK[1866] := 16#4ED8;
   // UNICODE_TO_GBK[1867] := 16#B8B6;
   // UNICODE_TO_GBK[1868] := 16#4ED9;
   // UNICODE_TO_GBK[1869] := 16#CFC9;
   // UNICODE_TO_GBK[1870] := 16#4EDA;
   // UNICODE_TO_GBK[1871] := 16#8199;
   // UNICODE_TO_GBK[1872] := 16#4EDB;
   // UNICODE_TO_GBK[1873] := 16#819A;
   // UNICODE_TO_GBK[1874] := 16#4EDC;
   // UNICODE_TO_GBK[1875] := 16#819B;
   // UNICODE_TO_GBK[1876] := 16#4EDD;
   // UNICODE_TO_GBK[1877] := 16#D9DA;
   // UNICODE_TO_GBK[1878] := 16#4EDE;
   // UNICODE_TO_GBK[1879] := 16#D8F0;
   // UNICODE_TO_GBK[1880] := 16#4EDF;
   // UNICODE_TO_GBK[1881] := 16#C7AA;
   // UNICODE_TO_GBK[1882] := 16#4EE0;
   // UNICODE_TO_GBK[1883] := 16#819C;
   // UNICODE_TO_GBK[1884] := 16#4EE1;
   // UNICODE_TO_GBK[1885] := 16#D8EE;
   // UNICODE_TO_GBK[1886] := 16#4EE2;
   // UNICODE_TO_GBK[1887] := 16#819D;
   // UNICODE_TO_GBK[1888] := 16#4EE3;
   // UNICODE_TO_GBK[1889] := 16#B4FA;
   // UNICODE_TO_GBK[1890] := 16#4EE4;
   // UNICODE_TO_GBK[1891] := 16#C1EE;
   // UNICODE_TO_GBK[1892] := 16#4EE5;
   // UNICODE_TO_GBK[1893] := 16#D2D4;
   // UNICODE_TO_GBK[1894] := 16#4EE6;
   // UNICODE_TO_GBK[1895] := 16#819E;
   // UNICODE_TO_GBK[1896] := 16#4EE7;
   // UNICODE_TO_GBK[1897] := 16#819F;
   // UNICODE_TO_GBK[1898] := 16#4EE8;
   // UNICODE_TO_GBK[1899] := 16#D8ED;
   // UNICODE_TO_GBK[1900] := 16#4EE9;
   // UNICODE_TO_GBK[1901] := 16#81A0;
   // UNICODE_TO_GBK[1902] := 16#4EEA;
   // UNICODE_TO_GBK[1903] := 16#D2C7;
   // UNICODE_TO_GBK[1904] := 16#4EEB;
   // UNICODE_TO_GBK[1905] := 16#D8EF;
   // UNICODE_TO_GBK[1906] := 16#4EEC;
   // UNICODE_TO_GBK[1907] := 16#C3C7;
   // UNICODE_TO_GBK[1908] := 16#4EED;
   // UNICODE_TO_GBK[1909] := 16#81A1;
   // UNICODE_TO_GBK[1910] := 16#4EEE;
   // UNICODE_TO_GBK[1911] := 16#81A2;
   // UNICODE_TO_GBK[1912] := 16#4EEF;
   // UNICODE_TO_GBK[1913] := 16#81A3;
   // UNICODE_TO_GBK[1914] := 16#4EF0;
   // UNICODE_TO_GBK[1915] := 16#D1F6;
   // UNICODE_TO_GBK[1916] := 16#4EF1;
   // UNICODE_TO_GBK[1917] := 16#81A4;
   // UNICODE_TO_GBK[1918] := 16#4EF2;
   // UNICODE_TO_GBK[1919] := 16#D6D9;
   // UNICODE_TO_GBK[1920] := 16#4EF3;
   // UNICODE_TO_GBK[1921] := 16#D8F2;
   // UNICODE_TO_GBK[1922] := 16#4EF4;
   // UNICODE_TO_GBK[1923] := 16#81A5;
   // UNICODE_TO_GBK[1924] := 16#4EF5;
   // UNICODE_TO_GBK[1925] := 16#D8F5;
   // UNICODE_TO_GBK[1926] := 16#4EF6;
   // UNICODE_TO_GBK[1927] := 16#BCFE;
   // UNICODE_TO_GBK[1928] := 16#4EF7;
   // UNICODE_TO_GBK[1929] := 16#BCDB;
   // UNICODE_TO_GBK[1930] := 16#4EF8;
   // UNICODE_TO_GBK[1931] := 16#81A6;
   // UNICODE_TO_GBK[1932] := 16#4EF9;
   // UNICODE_TO_GBK[1933] := 16#81A7;
   // UNICODE_TO_GBK[1934] := 16#4EFA;
   // UNICODE_TO_GBK[1935] := 16#81A8;
   // UNICODE_TO_GBK[1936] := 16#4EFB;
   // UNICODE_TO_GBK[1937] := 16#C8CE;
   // UNICODE_TO_GBK[1938] := 16#4EFC;
   // UNICODE_TO_GBK[1939] := 16#81A9;
   // UNICODE_TO_GBK[1940] := 16#4EFD;
   // UNICODE_TO_GBK[1941] := 16#B7DD;
   // UNICODE_TO_GBK[1942] := 16#4EFE;
   // UNICODE_TO_GBK[1943] := 16#81AA;
   // UNICODE_TO_GBK[1944] := 16#4EFF;
   // UNICODE_TO_GBK[1945] := 16#B7C2;
   // UNICODE_TO_GBK[1946] := 16#4F00;
   // UNICODE_TO_GBK[1947] := 16#81AB;
   // UNICODE_TO_GBK[1948] := 16#4F01;
   // UNICODE_TO_GBK[1949] := 16#C6F3;
   // UNICODE_TO_GBK[1950] := 16#4F02;
   // UNICODE_TO_GBK[1951] := 16#81AC;
   // UNICODE_TO_GBK[1952] := 16#4F03;
   // UNICODE_TO_GBK[1953] := 16#81AD;
   // UNICODE_TO_GBK[1954] := 16#4F04;
   // UNICODE_TO_GBK[1955] := 16#81AE;
   // UNICODE_TO_GBK[1956] := 16#4F05;
   // UNICODE_TO_GBK[1957] := 16#81AF;
   // UNICODE_TO_GBK[1958] := 16#4F06;
   // UNICODE_TO_GBK[1959] := 16#81B0;
   // UNICODE_TO_GBK[1960] := 16#4F07;
   // UNICODE_TO_GBK[1961] := 16#81B1;
   // UNICODE_TO_GBK[1962] := 16#4F08;
   // UNICODE_TO_GBK[1963] := 16#81B2;
   // UNICODE_TO_GBK[1964] := 16#4F09;
   // UNICODE_TO_GBK[1965] := 16#D8F8;
   // UNICODE_TO_GBK[1966] := 16#4F0A;
   // UNICODE_TO_GBK[1967] := 16#D2C1;
   // UNICODE_TO_GBK[1968] := 16#4F0B;
   // UNICODE_TO_GBK[1969] := 16#81B3;
   // UNICODE_TO_GBK[1970] := 16#4F0C;
   // UNICODE_TO_GBK[1971] := 16#81B4;
   // UNICODE_TO_GBK[1972] := 16#4F0D;
   // UNICODE_TO_GBK[1973] := 16#CEE9;
   // UNICODE_TO_GBK[1974] := 16#4F0E;
   // UNICODE_TO_GBK[1975] := 16#BCBF;
   // UNICODE_TO_GBK[1976] := 16#4F0F;
   // UNICODE_TO_GBK[1977] := 16#B7FC;
   // UNICODE_TO_GBK[1978] := 16#4F10;
   // UNICODE_TO_GBK[1979] := 16#B7A5;
   // UNICODE_TO_GBK[1980] := 16#4F11;
   // UNICODE_TO_GBK[1981] := 16#D0DD;
   // UNICODE_TO_GBK[1982] := 16#4F12;
   // UNICODE_TO_GBK[1983] := 16#81B5;
   // UNICODE_TO_GBK[1984] := 16#4F13;
   // UNICODE_TO_GBK[1985] := 16#81B6;
   // UNICODE_TO_GBK[1986] := 16#4F14;
   // UNICODE_TO_GBK[1987] := 16#81B7;
   // UNICODE_TO_GBK[1988] := 16#4F15;
   // UNICODE_TO_GBK[1989] := 16#81B8;
   // UNICODE_TO_GBK[1990] := 16#4F16;
   // UNICODE_TO_GBK[1991] := 16#81B9;
   // UNICODE_TO_GBK[1992] := 16#4F17;
   // UNICODE_TO_GBK[1993] := 16#D6DA;
   // UNICODE_TO_GBK[1994] := 16#4F18;
   // UNICODE_TO_GBK[1995] := 16#D3C5;
   // UNICODE_TO_GBK[1996] := 16#4F19;
   // UNICODE_TO_GBK[1997] := 16#BBEF;
   // UNICODE_TO_GBK[1998] := 16#4F1A;
   // UNICODE_TO_GBK[1999] := 16#BBE1;
   // UNICODE_TO_GBK[2000] := 16#4F1B;
   // UNICODE_TO_GBK[2001] := 16#D8F1;
   // UNICODE_TO_GBK[2002] := 16#4F1C;
   // UNICODE_TO_GBK[2003] := 16#81BA;
   // UNICODE_TO_GBK[2004] := 16#4F1D;
   // UNICODE_TO_GBK[2005] := 16#81BB;
   // UNICODE_TO_GBK[2006] := 16#4F1E;
   // UNICODE_TO_GBK[2007] := 16#C9A1;
   // UNICODE_TO_GBK[2008] := 16#4F1F;
   // UNICODE_TO_GBK[2009] := 16#CEB0;
   // UNICODE_TO_GBK[2010] := 16#4F20;
   // UNICODE_TO_GBK[2011] := 16#B4AB;
   // UNICODE_TO_GBK[2012] := 16#4F21;
   // UNICODE_TO_GBK[2013] := 16#81BC;
   // UNICODE_TO_GBK[2014] := 16#4F22;
   // UNICODE_TO_GBK[2015] := 16#D8F3;
   // UNICODE_TO_GBK[2016] := 16#4F23;
   // UNICODE_TO_GBK[2017] := 16#81BD;
   // UNICODE_TO_GBK[2018] := 16#4F24;
   // UNICODE_TO_GBK[2019] := 16#C9CB;
   // UNICODE_TO_GBK[2020] := 16#4F25;
   // UNICODE_TO_GBK[2021] := 16#D8F6;
   // UNICODE_TO_GBK[2022] := 16#4F26;
   // UNICODE_TO_GBK[2023] := 16#C2D7;
   // UNICODE_TO_GBK[2024] := 16#4F27;
   // UNICODE_TO_GBK[2025] := 16#D8F7;
   // UNICODE_TO_GBK[2026] := 16#4F28;
   // UNICODE_TO_GBK[2027] := 16#81BE;
   // UNICODE_TO_GBK[2028] := 16#4F29;
   // UNICODE_TO_GBK[2029] := 16#81BF;
   // UNICODE_TO_GBK[2030] := 16#4F2A;
   // UNICODE_TO_GBK[2031] := 16#CEB1;
   // UNICODE_TO_GBK[2032] := 16#4F2B;
   // UNICODE_TO_GBK[2033] := 16#D8F9;
   // UNICODE_TO_GBK[2034] := 16#4F2C;
   // UNICODE_TO_GBK[2035] := 16#81C0;
   // UNICODE_TO_GBK[2036] := 16#4F2D;
   // UNICODE_TO_GBK[2037] := 16#81C1;
   // UNICODE_TO_GBK[2038] := 16#4F2E;
   // UNICODE_TO_GBK[2039] := 16#81C2;
   // UNICODE_TO_GBK[2040] := 16#4F2F;
   // UNICODE_TO_GBK[2041] := 16#B2AE;
   // UNICODE_TO_GBK[2042] := 16#4F30;
   // UNICODE_TO_GBK[2043] := 16#B9C0;
   // UNICODE_TO_GBK[2044] := 16#4F31;
   // UNICODE_TO_GBK[2045] := 16#81C3;
   // UNICODE_TO_GBK[2046] := 16#4F32;
   // UNICODE_TO_GBK[2047] := 16#D9A3;
   // UNICODE_TO_GBK[2048] := 16#4F33;
   // UNICODE_TO_GBK[2049] := 16#81C4;
   // UNICODE_TO_GBK[2050] := 16#4F34;
   // UNICODE_TO_GBK[2051] := 16#B0E9;
   // UNICODE_TO_GBK[2052] := 16#4F35;
   // UNICODE_TO_GBK[2053] := 16#81C5;
   // UNICODE_TO_GBK[2054] := 16#4F36;
   // UNICODE_TO_GBK[2055] := 16#C1E6;
   // UNICODE_TO_GBK[2056] := 16#4F37;
   // UNICODE_TO_GBK[2057] := 16#81C6;
   // UNICODE_TO_GBK[2058] := 16#4F38;
   // UNICODE_TO_GBK[2059] := 16#C9EC;
   // UNICODE_TO_GBK[2060] := 16#4F39;
   // UNICODE_TO_GBK[2061] := 16#81C7;
   // UNICODE_TO_GBK[2062] := 16#4F3A;
   // UNICODE_TO_GBK[2063] := 16#CBC5;
   // UNICODE_TO_GBK[2064] := 16#4F3B;
   // UNICODE_TO_GBK[2065] := 16#81C8;
   // UNICODE_TO_GBK[2066] := 16#4F3C;
   // UNICODE_TO_GBK[2067] := 16#CBC6;
   // UNICODE_TO_GBK[2068] := 16#4F3D;
   // UNICODE_TO_GBK[2069] := 16#D9A4;
   // UNICODE_TO_GBK[2070] := 16#4F3E;
   // UNICODE_TO_GBK[2071] := 16#81C9;
   // UNICODE_TO_GBK[2072] := 16#4F3F;
   // UNICODE_TO_GBK[2073] := 16#81CA;
   // UNICODE_TO_GBK[2074] := 16#4F40;
   // UNICODE_TO_GBK[2075] := 16#81CB;
   // UNICODE_TO_GBK[2076] := 16#4F41;
   // UNICODE_TO_GBK[2077] := 16#81CC;
   // UNICODE_TO_GBK[2078] := 16#4F42;
   // UNICODE_TO_GBK[2079] := 16#81CD;
   // UNICODE_TO_GBK[2080] := 16#4F43;
   // UNICODE_TO_GBK[2081] := 16#B5E8;
   // UNICODE_TO_GBK[2082] := 16#4F44;
   // UNICODE_TO_GBK[2083] := 16#81CE;
   // UNICODE_TO_GBK[2084] := 16#4F45;
   // UNICODE_TO_GBK[2085] := 16#81CF;
   // UNICODE_TO_GBK[2086] := 16#4F46;
   // UNICODE_TO_GBK[2087] := 16#B5AB;
   // UNICODE_TO_GBK[2088] := 16#4F47;
   // UNICODE_TO_GBK[2089] := 16#81D0;
   // UNICODE_TO_GBK[2090] := 16#4F48;
   // UNICODE_TO_GBK[2091] := 16#81D1;
   // UNICODE_TO_GBK[2092] := 16#4F49;
   // UNICODE_TO_GBK[2093] := 16#81D2;
   // UNICODE_TO_GBK[2094] := 16#4F4A;
   // UNICODE_TO_GBK[2095] := 16#81D3;
   // UNICODE_TO_GBK[2096] := 16#4F4B;
   // UNICODE_TO_GBK[2097] := 16#81D4;
   // UNICODE_TO_GBK[2098] := 16#4F4C;
   // UNICODE_TO_GBK[2099] := 16#81D5;
   // UNICODE_TO_GBK[2100] := 16#4F4D;
   // UNICODE_TO_GBK[2101] := 16#CEBB;
   // UNICODE_TO_GBK[2102] := 16#4F4E;
   // UNICODE_TO_GBK[2103] := 16#B5CD;
   // UNICODE_TO_GBK[2104] := 16#4F4F;
   // UNICODE_TO_GBK[2105] := 16#D7A1;
   // UNICODE_TO_GBK[2106] := 16#4F50;
   // UNICODE_TO_GBK[2107] := 16#D7F4;
   // UNICODE_TO_GBK[2108] := 16#4F51;
   // UNICODE_TO_GBK[2109] := 16#D3D3;
   // UNICODE_TO_GBK[2110] := 16#4F52;
   // UNICODE_TO_GBK[2111] := 16#81D6;
   // UNICODE_TO_GBK[2112] := 16#4F53;
   // UNICODE_TO_GBK[2113] := 16#CCE5;
   // UNICODE_TO_GBK[2114] := 16#4F54;
   // UNICODE_TO_GBK[2115] := 16#81D7;
   // UNICODE_TO_GBK[2116] := 16#4F55;
   // UNICODE_TO_GBK[2117] := 16#BACE;
   // UNICODE_TO_GBK[2118] := 16#4F56;
   // UNICODE_TO_GBK[2119] := 16#81D8;
   // UNICODE_TO_GBK[2120] := 16#4F57;
   // UNICODE_TO_GBK[2121] := 16#D9A2;
   // UNICODE_TO_GBK[2122] := 16#4F58;
   // UNICODE_TO_GBK[2123] := 16#D9DC;
   // UNICODE_TO_GBK[2124] := 16#4F59;
   // UNICODE_TO_GBK[2125] := 16#D3E0;
   // UNICODE_TO_GBK[2126] := 16#4F5A;
   // UNICODE_TO_GBK[2127] := 16#D8FD;
   // UNICODE_TO_GBK[2128] := 16#4F5B;
   // UNICODE_TO_GBK[2129] := 16#B7F0;
